C05483=1150.206,331.149,-77.116,-176.637,8.840,148.788
C05484=1150.202,331.397,-77.150,-176.634,8.844,148.788
C05485=1150.198,331.645,-77.183,-176.632,8.847,148.789
C05486=1150.193,331.893,-77.216,-176.629,8.851,148.789
C05487=1150.190,332.140,-77.248,-176.627,8.854,148.789
C05488=1150.186,332.388,-77.282,-176.624,8.858,148.789
C05489=1150.182,332.635,-77.315,-176.621,8.862,148.789
C05490=1150.178,332.883,-77.348,-176.619,8.865,148.790
C05491=1150.174,333.131,-77.381,-176.616,8.869,148.790
C05492=1150.169,333.379,-77.414,-176.614,8.872,148.790
C05493=1150.165,333.626,-77.447,-176.611,8.877,148.790
C05494=1150.161,333.874,-77.481,-176.609,8.880,148.791
C05495=1150.157,334.122,-77.514,-176.606,8.883,148.791
C05496=1150.153,334.370,-77.547,-176.603,8.887,148.791
C05497=1150.149,334.617,-77.580,-176.601,8.890,148.791
C05498=1150.145,334.865,-77.613,-176.599,8.895,148.792
C05499=1150.141,335.113,-77.647,-176.596,8.898,148.792
C05500=1150.137,335.361,-77.680,-176.593,8.902,148.792
C05501=1150.133,335.609,-77.713,-176.591,8.906,148.792
C05502=1150.129,335.856,-77.747,-176.589,8.909,148.792
C05503=1150.125,336.104,-77.780,-176.586,8.913,148.793
C05504=1150.121,336.351,-77.813,-176.583,8.916,148.793
C05505=1150.116,336.599,-77.846,-176.580,8.920,148.793
C05506=1150.112,336.847,-77.879,-176.578,8.924,148.793
C05507=1150.109,337.095,-77.913,-176.576,8.928,148.794
C05508=1150.105,337.342,-77.947,-176.573,8.931,148.794
C05509=1150.101,337.590,-77.980,-176.570,8.935,148.794
C05510=1150.097,337.838,-78.013,-176.568,8.939,148.794
C05511=1150.092,338.086,-78.047,-176.565,8.943,148.795
C05512=1150.088,338.333,-78.081,-176.563,8.946,148.795
C05513=1150.084,338.581,-78.114,-176.560,8.950,148.795
C05514=1150.080,338.829,-78.147,-176.558,8.953,148.795
C05515=1150.076,339.109,-78.185,-176.555,8.958,148.796
C05516=1150.071,339.389,-78.224,-176.552,8.962,148.796
C05517=1150.067,339.670,-78.261,-176.549,8.966,148.796
C05518=1150.062,339.950,-78.300,-176.547,8.970,148.797
C05519=1150.057,340.197,-78.333,-176.544,8.974,148.797
C05520=1150.054,340.445,-78.367,-176.541,8.977,148.797
C05521=1150.050,340.693,-78.400,-176.539,8.982,148.797
C05522=1150.046,340.940,-78.435,-176.536,8.985,148.798
C05523=1150.041,341.188,-78.468,-176.534,8.989,148.798
C05524=1150.038,341.436,-78.502,-176.531,8.992,148.798
C05525=1150.034,341.684,-78.535,-176.528,8.996,148.798
C05526=1150.029,341.931,-78.570,-176.526,9.000,148.799
C05527=1150.025,342.179,-78.603,-176.524,9.004,148.799
C05528=1150.022,342.427,-78.637,-176.521,9.007,148.799
C05529=1150.018,342.674,-78.670,-176.518,9.011,148.799
C05530=1150.013,342.922,-78.705,-176.516,9.015,148.800
C05531=1150.009,343.169,-78.738,-176.514,9.019,148.800
C05532=1150.006,343.417,-78.772,-176.511,9.022,148.800
C05533=1150.001,343.665,-78.806,-176.508,9.027,148.801
C05534=1149.997,343.912,-78.840,-176.506,9.030,148.801
C05535=1149.993,344.159,-78.873,-176.503,9.034,148.801
C05536=1149.989,344.408,-78.908,-176.501,9.037,148.801
C05537=1149.985,344.655,-78.941,-176.498,9.042,148.802
C05538=1149.981,344.903,-78.976,-176.496,9.045,148.802
C05539=1149.977,345.151,-79.009,-176.493,9.049,148.802
C05540=1149.973,345.398,-79.043,-176.491,9.052,148.803
C05541=1149.969,345.646,-79.078,-176.488,9.057,148.803
C05542=1149.965,345.894,-79.111,-176.486,9.060,148.803
C05543=1149.961,346.142,-79.146,-176.483,9.064,148.803
C05544=1149.957,346.389,-79.180,-176.481,9.068,148.804
C05545=1149.954,346.636,-79.214,-176.478,9.072,148.804
C05546=1149.949,346.884,-79.248,-176.476,9.075,148.804
C05547=1149.945,347.132,-79.281,-176.473,9.079,148.804
C05548=1149.941,347.380,-79.316,-176.471,9.083,148.805
C05549=1149.937,347.627,-79.350,-176.468,9.087,148.805
C05550=1149.933,347.875,-79.385,-176.466,9.090,148.805
C05551=1149.929,348.122,-79.419,-176.463,9.094,148.805
C05552=1149.925,348.370,-79.453,-176.461,9.098,148.806
C05553=1149.921,348.618,-79.487,-176.458,9.102,148.806
C05554=1149.917,348.865,-79.521,-176.455,9.106,148.806
C05555=1149.913,349.113,-79.556,-176.453,9.109,148.807
C05556=1149.909,349.361,-79.590,-176.450,9.113,148.807
C05557=1149.905,349.608,-79.624,-176.448,9.117,148.807
C05558=1149.901,349.856,-79.659,-176.445,9.121,148.808
C05559=1149.897,350.103,-79.693,-176.443,9.124,148.808
C05560=1149.893,350.351,-79.727,-176.440,9.128,148.808
C05561=1149.889,350.598,-79.761,-176.438,9.132,148.808
C05562=1149.886,350.846,-79.796,-176.436,9.136,148.809
C05563=1149.881,351.094,-79.831,-176.433,9.139,148.809
C05564=1149.878,351.341,-79.865,-176.430,9.144,148.809
C05565=1149.873,351.589,-79.899,-176.428,9.148,148.810
C05566=1149.869,351.836,-79.933,-176.426,9.151,148.810
C05567=1149.865,352.084,-79.968,-176.423,9.155,148.810
C05568=1149.861,352.332,-80.003,-176.421,9.159,148.811
C05569=1149.858,352.579,-80.037,-176.418,9.163,148.811
C05570=1149.853,352.826,-80.072,-176.416,9.166,148.811
C05571=1149.849,353.074,-80.107,-176.413,9.171,148.812
C05572=1149.845,353.321,-80.141,-176.410,9.175,148.812
C05573=1149.842,353.570,-80.175,-176.408,9.178,148.812
C05574=1149.837,353.817,-80.210,-176.405,9.182,148.813
C05575=1149.834,354.065,-80.244,-176.403,9.186,148.813
C05576=1149.830,354.312,-80.280,-176.400,9.190,148.813
C05577=1149.825,354.560,-80.314,-176.398,9.193,148.813
C05578=1149.822,354.808,-80.349,-176.395,9.197,148.814
C05579=1149.818,355.055,-80.383,-176.393,9.202,148.814
C05580=1149.814,355.302,-80.418,-176.391,9.205,148.814
C05581=1149.809,355.550,-80.453,-176.388,9.209,148.815
C05582=1149.806,355.798,-80.487,-176.386,9.213,148.815
C05583=1149.802,356.044,-80.522,-176.383,9.217,148.815
C05584=1149.798,356.293,-80.557,-176.380,9.221,148.816
C05585=1149.794,356.541,-80.592,-176.378,9.225,148.816
C05586=1149.790,356.787,-80.627,-176.375,9.229,148.816
C05587=1149.787,357.035,-80.661,-176.373,9.232,148.817
C05588=1149.782,357.282,-80.697,-176.370,9.236,148.817
C05589=1149.778,357.530,-80.731,-176.367,9.240,148.817
C05590=1149.774,357.778,-80.766,-176.365,9.244,148.818
C05591=1149.770,358.025,-80.801,-176.363,9.248,148.818
C05592=1149.767,358.273,-80.836,-176.361,9.252,148.818
C05593=1149.763,358.520,-80.871,-176.358,9.256,148.818
C05594=1149.759,358.768,-80.906,-176.355,9.260,148.819
C05595=1149.755,359.015,-80.941,-176.353,9.263,148.819
C05596=1149.750,359.263,-80.976,-176.350,9.267,148.819
C05597=1149.747,359.510,-81.011,-176.348,9.272,148.820
C05598=1149.743,359.758,-81.046,-176.345,9.275,148.820
C05599=1149.738,360.005,-81.081,-176.342,9.279,148.820
C05600=1149.735,360.253,-81.117,-176.340,9.284,148.821
C05601=1149.732,360.500,-81.151,-176.338,9.287,148.821
C05602=1149.727,360.747,-81.186,-176.335,9.291,148.821
C05603=1149.723,360.995,-81.221,-176.332,9.295,148.822
C05604=1149.720,361.243,-81.257,-176.330,9.299,148.822
C05605=1149.715,361.490,-81.292,-176.327,9.303,148.822
C05606=1149.711,361.738,-81.327,-176.324,9.307,148.823
C05607=1149.708,361.985,-81.362,-176.322,9.312,148.823
C05608=1149.704,362.233,-81.398,-176.320,9.315,148.823
C05609=1149.700,362.480,-81.433,-176.317,9.319,148.824
C05610=1149.696,362.728,-81.468,-176.314,9.323,148.824
C05611=1149.692,362.975,-81.503,-176.312,9.327,148.824
C05612=1149.688,363.222,-81.538,-176.309,9.331,148.825
C05613=1149.684,363.470,-81.574,-176.306,9.335,148.825
C05614=1149.680,363.718,-81.609,-176.304,9.339,148.825
C05615=1149.677,363.965,-81.644,-176.302,9.343,148.826
C05616=1149.673,364.213,-81.680,-176.299,9.347,148.826
C05617=1149.669,364.459,-81.715,-176.296,9.351,148.826
C05618=1149.665,364.707,-81.751,-176.293,9.355,148.827
C05619=1149.661,364.990,-81.791,-176.291,9.360,148.827
C05620=1149.656,365.274,-81.832,-176.287,9.365,148.828
C05621=1149.651,365.556,-81.873,-176.285,9.369,148.828
C05622=1149.646,365.840,-81.913,-176.281,9.374,148.828
C05623=1149.643,366.088,-81.948,-176.280,9.377,148.829
C05624=1149.639,366.335,-81.984,-176.277,9.382,148.829
C05625=1149.636,366.583,-82.019,-176.274,9.386,148.829
C05626=1149.631,366.830,-82.055,-176.271,9.390,148.830
C05627=1149.627,367.077,-82.091,-176.269,9.394,148.830
C05628=1149.623,367.325,-82.126,-176.266,9.398,148.830
C05629=1149.620,367.572,-82.162,-176.264,9.402,148.831
C05630=1149.616,367.820,-82.197,-176.261,9.407,148.831
C05631=1149.613,368.067,-82.234,-176.259,9.411,148.832
C05632=1149.608,368.314,-82.269,-176.257,9.414,148.832
C05633=1149.604,368.561,-82.305,-176.254,9.418,148.832
C05634=1149.600,368.809,-82.340,-176.251,9.423,148.833
C05635=1149.597,369.056,-82.376,-176.249,9.427,148.833
C05636=1149.592,369.304,-82.412,-176.246,9.430,148.833
C05637=1149.588,369.552,-82.448,-176.244,9.435,148.834
C05638=1149.585,369.799,-82.483,-176.241,9.439,148.834
C05639=1149.581,370.046,-82.520,-176.239,9.443,148.835
C05640=1149.576,370.293,-82.555,-176.236,9.448,148.835
C05641=1149.573,370.541,-82.591,-176.234,9.451,148.836
C05642=1149.569,370.788,-82.626,-176.232,9.456,148.836
C05643=1149.565,371.036,-82.663,-176.229,9.460,148.837
C05644=1149.561,371.283,-82.699,-176.226,9.464,148.837
C05645=1149.558,371.530,-82.734,-176.224,9.468,148.837
C05646=1149.553,371.778,-82.770,-176.222,9.472,148.838
C05647=1149.550,372.025,-82.807,-176.219,9.476,148.838
C05648=1149.546,372.273,-82.843,-176.217,9.480,148.839
C05649=1149.542,372.520,-82.878,-176.215,9.484,148.839
C05650=1149.539,372.767,-82.915,-176.212,9.489,148.840
C05651=1149.534,373.015,-82.951,-176.211,9.492,148.840
C05652=1149.530,373.263,-82.986,-176.208,9.497,148.840
C05653=1149.527,373.510,-83.023,-176.206,9.501,148.841
C05654=1149.523,373.757,-83.059,-176.204,9.505,148.841
C05655=1149.519,374.004,-83.095,-176.201,9.509,148.842
C05656=1149.515,374.252,-83.131,-176.199,9.514,148.842
C05657=1149.511,374.498,-83.167,-176.197,9.517,148.843
C05658=1149.507,374.746,-83.203,-176.195,9.522,148.843
C05659=1149.503,374.994,-83.239,-176.193,9.525,148.844
C05660=1149.499,375.241,-83.276,-176.191,9.530,148.844
C05661=1149.495,375.488,-83.311,-176.189,9.534,148.845
C05662=1149.492,375.736,-83.348,-176.186,9.538,148.845
C05663=1149.488,375.983,-83.385,-176.185,9.542,148.846
C05664=1149.484,376.231,-83.421,-176.182,9.546,148.846
C05665=1149.481,376.478,-83.457,-176.181,9.550,148.847
C05666=1149.476,376.726,-83.493,-176.178,9.555,148.848
C05667=1149.473,376.972,-83.529,-176.177,9.559,148.848
C05668=1149.468,377.220,-83.566,-176.175,9.562,148.849
C05669=1149.465,377.467,-83.602,-176.173,9.567,148.849
C05670=1149.461,377.714,-83.639,-176.172,9.571,148.850
C05671=1149.457,377.962,-83.674,-176.170,9.574,148.850
C05672=1149.453,378.209,-83.711,-176.168,9.579,148.851
C05673=1149.449,378.456,-83.748,-176.166,9.583,148.852
C05674=1149.445,378.704,-83.784,-176.165,9.587,148.852
C05675=1149.441,378.951,-83.820,-176.163,9.591,148.853
C05676=1149.438,379.198,-83.857,-176.162,9.595,148.853
C05677=1149.434,379.446,-83.893,-176.160,9.598,148.854
C05678=1149.429,379.693,-83.930,-176.159,9.602,148.855
C05679=1149.426,379.940,-83.966,-176.157,9.607,148.855
C05680=1149.422,380.187,-84.003,-176.155,9.611,148.856
C05681=1149.419,380.435,-84.039,-176.154,9.614,148.856
C05682=1149.415,380.682,-84.076,-176.153,9.618,148.857
C05683=1149.411,380.929,-84.112,-176.152,9.622,148.858
C05684=1149.407,381.176,-84.149,-176.150,9.626,148.859
C05685=1149.403,381.423,-84.186,-176.149,9.630,148.859
C05686=1149.399,381.671,-84.222,-176.148,9.634,148.860
C05687=1149.396,381.918,-84.258,-176.147,9.637,148.861
C05688=1149.391,382.165,-84.295,-176.146,9.641,148.861
C05689=1149.387,382.413,-84.332,-176.145,9.644,148.862
C05690=1149.385,382.660,-84.368,-176.144,9.649,148.863
C05691=1149.381,382.907,-84.405,-176.143,9.652,148.863
C05692=1149.376,383.154,-84.442,-176.142,9.656,148.864
C05693=1149.372,383.402,-84.478,-176.141,9.659,148.865
C05694=1149.369,383.649,-84.514,-176.140,9.663,148.866
C05695=1149.365,383.896,-84.551,-176.140,9.667,148.866
C05696=1149.360,384.144,-84.588,-176.139,9.670,148.867
C05697=1149.358,384.391,-84.625,-176.138,9.673,148.868
C05698=1149.354,384.638,-84.662,-176.138,9.677,148.868
C05699=1149.350,384.886,-84.699,-176.137,9.680,148.869
C05700=1149.345,385.133,-84.735,-176.137,9.684,148.870
C05701=1149.342,385.380,-84.772,-176.137,9.687,148.871
C05702=1149.338,385.627,-84.808,-176.136,9.690,148.872
C05703=1149.335,385.875,-84.846,-176.136,9.694,148.872
C05704=1149.330,386.122,-84.883,-176.136,9.696,148.873
C05705=1149.327,386.369,-84.919,-176.136,9.700,148.874
C05706=1149.323,386.616,-84.956,-176.136,9.703,148.875
C05707=1149.319,386.863,-84.993,-176.136,9.706,148.876
C05708=1149.315,387.111,-85.030,-176.136,9.710,148.877
C05709=1149.311,387.358,-85.067,-176.136,9.712,148.877
C05710=1149.308,387.605,-85.103,-176.136,9.715,148.878
C05711=1149.304,387.852,-85.140,-176.136,9.719,148.879
C05712=1149.300,388.099,-85.177,-176.136,9.721,148.880
C05713=1149.296,388.347,-85.214,-176.136,9.724,148.880
C05714=1149.293,388.594,-85.250,-176.137,9.727,148.881
C05715=1149.289,388.841,-85.287,-176.136,9.730,148.882
C05716=1149.285,389.089,-85.324,-176.137,9.733,148.883
C05717=1149.281,389.336,-85.361,-176.138,9.736,148.884
C05718=1149.277,389.584,-85.398,-176.138,9.739,148.885
C05719=1149.274,389.831,-85.434,-176.138,9.741,148.886
C05720=1149.270,390.078,-85.471,-176.139,9.744,148.886
C05721=1149.266,390.325,-85.508,-176.139,9.747,148.887
C05722=1149.261,390.572,-85.545,-176.140,9.749,148.888
C05723=1149.257,390.858,-85.588,-176.141,9.752,148.889
C05724=1149.253,391.145,-85.630,-176.141,9.755,148.890
C05725=1149.249,391.432,-85.673,-176.142,9.758,148.891
C05726=1149.244,391.718,-85.716,-176.143,9.761,148.892
C05727=1149.241,391.966,-85.753,-176.143,9.764,148.893
C05728=1149.237,392.213,-85.790,-176.144,9.767,148.894
C05729=1149.233,392.460,-85.827,-176.145,9.769,148.895
C05730=1149.229,392.707,-85.863,-176.145,9.771,148.895
C05731=1149.225,392.955,-85.900,-176.146,9.773,148.896
C05732=1149.222,393.202,-85.937,-176.147,9.776,148.897
C05733=1149.218,393.449,-85.974,-176.148,9.778,148.898
C05734=1149.214,393.696,-86.011,-176.148,9.781,148.899
C05735=1149.210,393.943,-86.048,-176.149,9.783,148.900
C05736=1149.206,394.191,-86.085,-176.151,9.785,148.900
C05737=1149.202,394.438,-86.122,-176.151,9.788,148.901
C05738=1149.199,394.685,-86.159,-176.152,9.790,148.902
C05739=1149.195,394.932,-86.195,-176.153,9.792,148.903
C05740=1149.191,395.180,-86.232,-176.153,9.795,148.904
C05741=1149.187,395.427,-86.269,-176.155,9.797,148.905
C05742=1149.183,395.675,-86.306,-176.156,9.799,148.905
C05743=1149.179,395.922,-86.343,-176.157,9.801,148.906
C05744=1149.175,396.168,-86.381,-176.157,9.804,148.907
C05745=1149.172,396.415,-86.417,-176.158,9.806,148.908
C05746=1149.168,396.663,-86.454,-176.160,9.808,148.909
C05747=1149.164,396.910,-86.491,-176.161,9.810,148.910
C05748=1149.160,397.158,-86.528,-176.162,9.812,148.910
C05749=1149.156,397.405,-86.565,-176.163,9.814,148.911
C05750=1149.153,397.653,-86.602,-176.164,9.816,148.912
C05751=1149.149,397.899,-86.638,-176.165,9.818,148.913
C05752=1149.145,398.147,-86.675,-176.166,9.820,148.914
C05753=1149.141,398.393,-86.713,-176.167,9.822,148.914
C05754=1149.137,398.640,-86.750,-176.167,9.825,148.915
C05755=1149.134,398.888,-86.787,-176.168,9.827,148.916
C05756=1149.130,399.135,-86.824,-176.170,9.829,148.917
C05757=1149.126,399.383,-86.861,-176.171,9.831,148.918
C05758=1149.122,399.630,-86.897,-176.172,9.833,148.919
C05759=1149.119,399.877,-86.934,-176.172,9.835,148.919
C05760=1149.115,400.125,-86.971,-176.174,9.836,148.920
C05761=1149.111,400.372,-87.008,-176.175,9.838,148.921
C05762=1149.107,400.618,-87.045,-176.176,9.840,148.922
C05763=1149.103,400.866,-87.082,-176.177,9.843,148.923
C05764=1149.099,401.113,-87.119,-176.179,9.845,148.923
C05765=1149.096,401.360,-87.156,-176.179,9.846,148.924
C05766=1149.092,401.608,-87.193,-176.180,9.848,148.925
C05767=1149.088,401.855,-87.229,-176.181,9.850,148.926
C05768=1149.084,402.102,-87.266,-176.183,9.853,148.927
C05769=1149.080,402.350,-87.303,-176.183,9.854,148.927
C05770=1149.076,402.596,-87.341,-176.184,9.856,148.928
C05771=1149.072,402.844,-87.378,-176.185,9.858,148.929
C05772=1149.069,403.090,-87.414,-176.187,9.860,148.930
C05773=1149.065,403.338,-87.451,-176.187,9.862,148.930
C05774=1149.061,403.586,-87.488,-176.189,9.863,148.931
C05775=1149.057,403.833,-87.525,-176.190,9.866,148.932
C05776=1149.053,404.080,-87.562,-176.191,9.867,148.933
C05777=1149.049,404.327,-87.599,-176.192,9.869,148.933
C05778=1149.045,404.575,-87.636,-176.193,9.871,148.934
C05779=1149.042,404.821,-87.673,-176.194,9.873,148.935
C05780=1149.038,405.068,-87.710,-176.195,9.875,148.936
C05781=1149.034,405.316,-87.747,-176.196,9.877,148.937
C05782=1149.031,405.564,-87.784,-176.196,9.879,148.937
C05783=1149.027,405.811,-87.821,-176.198,9.881,148.938
C05784=1149.023,406.058,-87.858,-176.199,9.882,148.939
C05785=1149.018,406.305,-87.895,-176.200,9.884,148.940
C05786=1149.015,406.552,-87.931,-176.201,9.886,148.940
C05787=1149.012,406.799,-87.969,-176.202,9.888,148.941
C05788=1149.008,407.046,-88.006,-176.203,9.890,148.942
C05789=1149.004,407.294,-88.042,-176.203,9.892,148.942
C05790=1149.000,407.541,-88.079,-176.205,9.894,148.943
C05791=1148.996,407.789,-88.117,-176.205,9.896,148.944
C05792=1148.992,408.036,-88.153,-176.206,9.898,148.945
C05793=1148.989,408.283,-88.190,-176.207,9.899,148.945
C05794=1148.985,408.530,-88.227,-176.208,9.901,148.946
C05795=1148.981,408.777,-88.264,-176.209,9.903,148.947
C05796=1148.977,409.024,-88.301,-176.209,9.905,148.948
C05797=1148.973,409.272,-88.338,-176.211,9.907,148.948
C05798=1148.969,409.519,-88.375,-176.211,9.909,148.949
C05799=1148.965,409.766,-88.412,-176.212,9.911,148.950
C05800=1148.962,410.014,-88.449,-176.213,9.913,148.951
C05801=1148.958,410.261,-88.485,-176.214,9.914,148.951
C05802=1148.954,410.508,-88.522,-176.215,9.916,148.952
C05803=1148.950,410.755,-88.560,-176.215,9.918,148.953
C05804=1148.947,411.002,-88.597,-176.216,9.920,148.953
C05805=1148.943,411.250,-88.634,-176.217,9.922,148.954
C05806=1148.939,411.497,-88.671,-176.218,9.924,148.955
C05807=1148.934,411.744,-88.708,-176.219,9.925,148.955
C05808=1148.931,411.991,-88.744,-176.220,9.928,148.956
C05809=1148.928,412.239,-88.781,-176.220,9.929,148.957
C05810=1148.924,412.485,-88.819,-176.221,9.931,148.957
C05811=1148.920,412.733,-88.856,-176.222,9.933,148.958
C05812=1148.916,412.980,-88.892,-176.223,9.935,148.959
C05813=1148.912,413.228,-88.930,-176.223,9.937,148.960
C05814=1148.908,413.475,-88.966,-176.224,9.939,148.960
C05815=1148.904,413.722,-89.003,-176.225,9.941,148.961
C05816=1148.901,413.969,-89.040,-176.225,9.943,148.962
C05817=1148.897,414.215,-89.077,-176.226,9.945,148.962
C05818=1148.893,414.463,-89.114,-176.227,9.946,148.963
C05819=1148.889,414.711,-89.151,-176.228,9.949,148.964
C05820=1148.886,414.958,-89.188,-176.228,9.950,148.965
C05821=1148.883,415.204,-89.225,-176.228,9.953,148.965
C05822=1148.881,415.453,-89.262,-176.229,9.955,148.966
C05823=1148.881,415.679,-89.296,-176.230,9.956,148.966
C05824=1148.880,415.906,-89.329,-176.231,9.958,148.967
C05825=1148.880,416.132,-89.362,-176.231,9.960,148.968
C05826=1148.881,416.359,-89.396,-176.231,9.961,148.968
C05827=1148.882,416.585,-89.429,-176.232,9.963,148.969
C05828=1148.885,416.812,-89.463,-176.233,9.965,148.969
C05829=1148.887,417.038,-89.495,-176.233,9.966,148.970
C05830=1148.891,417.263,-89.528,-176.234,9.968,148.971
C05831=1148.470,417.266,-89.578,-176.236,9.979,148.974
C05832=1148.467,417.038,-89.545,-176.236,9.977,148.973
C05833=1148.464,416.810,-89.511,-176.235,9.975,148.973
C05834=1148.462,416.582,-89.478,-176.235,9.974,148.972
C05835=1148.460,416.354,-89.444,-176.234,9.972,148.972
C05836=1148.460,416.126,-89.410,-176.233,9.970,148.971
C05837=1148.460,415.897,-89.376,-176.233,9.969,148.971
C05838=1148.460,415.669,-89.342,-176.232,9.967,148.970
C05839=1148.461,415.441,-89.309,-176.232,9.965,148.969
C05840=1148.463,415.194,-89.272,-176.231,9.964,148.969
C05841=1148.465,414.946,-89.236,-176.230,9.962,148.968
C05842=1148.469,414.699,-89.198,-176.229,9.960,148.967
C05843=1148.473,414.452,-89.161,-176.229,9.958,148.967
C05844=1148.476,414.204,-89.124,-176.229,9.955,148.966
C05845=1148.480,413.957,-89.087,-176.228,9.954,148.965
C05846=1148.484,413.710,-89.051,-176.227,9.952,148.964
C05847=1148.488,413.463,-89.014,-176.226,9.950,148.964
C05848=1148.492,413.216,-88.976,-176.225,9.948,148.963
C05849=1148.495,412.968,-88.939,-176.224,9.946,148.962
C05850=1148.499,412.721,-88.902,-176.224,9.944,148.962
C05851=1148.503,412.474,-88.865,-176.223,9.943,148.961
C05852=1148.507,412.227,-88.828,-176.223,9.940,148.960
C05853=1148.510,411.979,-88.792,-176.222,9.938,148.960
C05854=1148.514,411.732,-88.755,-176.221,9.936,148.959
C05855=1148.518,411.485,-88.717,-176.221,9.934,148.958
C05856=1148.522,411.238,-88.680,-176.219,9.932,148.957
C05857=1148.526,410.990,-88.643,-176.219,9.931,148.957
C05858=1148.530,410.743,-88.606,-176.218,9.929,148.956
C05859=1148.534,410.496,-88.569,-176.217,9.927,148.955
C05860=1148.538,410.249,-88.533,-176.216,9.925,148.955
C05861=1148.541,410.003,-88.496,-176.215,9.923,148.954
C05862=1148.544,409.755,-88.458,-176.215,9.921,148.953
C05863=1148.548,409.507,-88.422,-176.213,9.919,148.952
C05864=1148.553,409.260,-88.385,-176.213,9.917,148.952
C05865=1148.557,409.013,-88.348,-176.212,9.916,148.951
C05866=1148.560,408.765,-88.311,-176.211,9.914,148.950
C05867=1148.564,408.518,-88.274,-176.210,9.912,148.950
C05868=1148.568,408.271,-88.236,-176.209,9.910,148.949
C05869=1148.571,408.025,-88.200,-176.209,9.908,148.948
C05870=1148.575,407.777,-88.163,-176.207,9.906,148.947
C05871=1148.579,407.530,-88.126,-176.207,9.904,148.947
C05872=1148.583,407.282,-88.089,-176.206,9.902,148.946
C05873=1148.587,407.035,-88.052,-176.205,9.900,148.945
C05874=1148.591,406.788,-88.015,-176.203,9.899,148.944
C05875=1148.595,406.540,-87.978,-176.202,9.897,148.944
C05876=1148.598,406.294,-87.941,-176.202,9.895,148.943
C05877=1148.602,406.047,-87.904,-176.200,9.893,148.942
C05878=1148.606,405.799,-87.867,-176.200,9.891,148.941
C05879=1148.610,405.552,-87.830,-176.199,9.889,148.941
C05880=1148.614,405.304,-87.793,-176.198,9.887,148.940
C05881=1148.618,405.057,-87.756,-176.197,9.886,148.939
C05882=1148.622,404.810,-87.720,-176.196,9.884,148.938
C05883=1148.626,404.563,-87.682,-176.195,9.881,148.937
C05884=1148.628,404.316,-87.645,-176.193,9.881,148.937
C05885=1148.632,404.069,-87.608,-176.192,9.878,148.936
C05886=1148.637,403.821,-87.572,-176.191,9.876,148.935
C05887=1148.641,403.574,-87.535,-176.191,9.875,148.935
C05888=1148.644,403.326,-87.498,-176.189,9.873,148.934
C05889=1148.648,403.079,-87.461,-176.188,9.871,148.933
C05890=1148.652,402.833,-87.423,-176.188,9.869,148.932
C05891=1148.655,402.586,-87.387,-176.187,9.867,148.931
C05892=1148.659,402.338,-87.350,-176.185,9.865,148.931
C05893=1148.663,402.091,-87.313,-176.184,9.863,148.930
C05894=1148.667,401.843,-87.276,-176.183,9.861,148.929
C05895=1148.671,401.596,-87.239,-176.182,9.860,148.928
C05896=1148.675,401.349,-87.202,-176.181,9.858,148.927
C05897=1148.679,401.101,-87.165,-176.180,9.855,148.927
C05898=1148.682,400.855,-87.128,-176.179,9.853,148.926
C05899=1148.686,400.608,-87.091,-176.178,9.851,148.925
C05900=1148.690,400.361,-87.054,-176.177,9.850,148.924
C05901=1148.693,400.113,-87.017,-176.176,9.848,148.923
C05902=1148.698,399.865,-86.980,-176.175,9.845,148.923
C05903=1148.702,399.618,-86.943,-176.174,9.843,148.922
C05904=1148.706,399.371,-86.906,-176.172,9.841,148.921
C05905=1148.709,399.124,-86.870,-176.171,9.839,148.920
C05906=1148.712,398.877,-86.832,-176.170,9.837,148.919
C05907=1148.716,398.630,-86.795,-176.169,9.835,148.918
C05908=1148.720,398.383,-86.759,-176.168,9.833,148.918
C05909=1148.725,398.135,-86.722,-176.167,9.831,148.917
C05910=1148.728,397.887,-86.684,-176.166,9.829,148.916
C05911=1148.732,397.640,-86.648,-176.165,9.827,148.915
C05912=1148.736,397.393,-86.611,-176.164,9.825,148.914
C05913=1148.740,397.146,-86.574,-176.163,9.823,148.914
C05914=1148.743,396.900,-86.537,-176.162,9.821,148.913
C05915=1148.747,396.652,-86.500,-176.161,9.819,148.912
C05916=1148.751,396.405,-86.463,-176.160,9.816,148.911
C05917=1148.755,396.157,-86.426,-176.159,9.814,148.910
C05918=1148.759,395.910,-86.389,-176.158,9.812,148.909
C05919=1148.763,395.662,-86.352,-176.157,9.810,148.909
C05920=1148.766,395.415,-86.316,-176.156,9.808,148.908
C05921=1148.770,395.168,-86.279,-176.156,9.805,148.907
C05922=1148.774,394.922,-86.241,-176.155,9.803,148.906
C05923=1148.778,394.674,-86.204,-176.153,9.801,148.905
C05924=1148.781,394.427,-86.167,-176.152,9.799,148.904
C05925=1148.786,394.179,-86.130,-176.152,9.796,148.904
C05926=1148.789,393.932,-86.094,-176.151,9.794,148.903
C05927=1148.793,393.685,-86.057,-176.150,9.792,148.902
C05928=1148.797,393.437,-86.020,-176.149,9.789,148.901
C05929=1148.801,393.190,-85.983,-176.148,9.787,148.900
C05930=1148.805,392.943,-85.946,-176.147,9.784,148.899
C05931=1148.809,392.696,-85.909,-176.147,9.783,148.899
C05932=1148.813,392.449,-85.872,-176.146,9.780,148.898
C05933=1148.815,392.202,-85.835,-176.145,9.778,148.897
C05934=1148.819,391.954,-85.798,-176.145,9.775,148.896
C05935=1148.824,391.707,-85.761,-176.144,9.772,148.895
C05936=1148.828,391.420,-85.719,-176.144,9.769,148.894
C05937=1148.832,391.134,-85.676,-176.143,9.766,148.893
C05938=1148.837,390.847,-85.633,-176.142,9.763,148.892
C05939=1148.841,390.561,-85.590,-176.141,9.760,148.891
C05940=1148.845,390.314,-85.553,-176.140,9.758,148.891
C05941=1148.848,390.066,-85.516,-176.140,9.755,148.890
C05942=1148.852,389.819,-85.480,-176.139,9.752,148.889
C05943=1148.856,389.572,-85.443,-176.139,9.750,148.888
C05944=1148.860,389.325,-85.406,-176.139,9.747,148.887
C05945=1148.864,389.077,-85.369,-176.138,9.744,148.886
C05946=1148.867,388.830,-85.332,-176.138,9.741,148.886
C05947=1148.871,388.583,-85.296,-176.138,9.739,148.885
C05948=1148.875,388.336,-85.259,-176.138,9.735,148.884
C05949=1148.880,388.088,-85.222,-176.138,9.732,148.883
C05950=1148.883,387.841,-85.185,-176.137,9.729,148.882
C05951=1148.886,387.594,-85.148,-176.137,9.727,148.881
C05952=1148.891,387.346,-85.111,-176.137,9.723,148.880
C05953=1148.895,387.099,-85.075,-176.137,9.721,148.880
C05954=1148.899,386.852,-85.038,-176.137,9.717,148.879
C05955=1148.902,386.604,-85.001,-176.137,9.714,148.878
C05956=1148.906,386.357,-84.964,-176.137,9.711,148.877
C05957=1148.910,386.110,-84.927,-176.137,9.708,148.877
C05958=1148.914,385.863,-84.891,-176.137,9.705,148.876
C05959=1148.918,385.616,-84.854,-176.138,9.701,148.875
C05960=1148.921,385.369,-84.817,-176.138,9.698,148.874
C05961=1148.925,385.121,-84.780,-176.139,9.695,148.873
C05962=1148.929,384.874,-84.743,-176.139,9.691,148.873
C05963=1148.933,384.627,-84.706,-176.140,9.688,148.872
C05964=1148.936,384.380,-84.670,-176.140,9.684,148.871
C05965=1148.940,384.133,-84.633,-176.141,9.681,148.870
C05966=1148.944,383.885,-84.597,-176.141,9.678,148.870
C05967=1148.948,383.637,-84.559,-176.142,9.674,148.869
C05968=1148.951,383.391,-84.523,-176.143,9.670,148.868
C05969=1148.955,383.143,-84.486,-176.144,9.667,148.867
C05970=1148.959,382.896,-84.449,-176.144,9.664,148.867
C05971=1148.963,382.649,-84.413,-176.145,9.659,148.866
C05972=1148.967,382.401,-84.377,-176.146,9.656,148.865
C05973=1148.971,382.154,-84.340,-176.147,9.652,148.865
C05974=1148.975,381.906,-84.303,-176.149,9.648,148.864
C05975=1148.978,381.660,-84.267,-176.149,9.645,148.863
C05976=1148.982,381.412,-84.230,-176.150,9.641,148.863
C05977=1148.986,381.165,-84.193,-176.152,9.637,148.862
C05978=1148.990,380.918,-84.157,-176.153,9.633,148.861
C05979=1148.994,380.670,-84.120,-176.155,9.629,148.860
C05980=1148.998,380.423,-84.084,-176.155,9.626,148.860
C05981=1149.002,380.176,-84.047,-176.157,9.622,148.859
C05982=1149.005,379.928,-84.010,-176.158,9.618,148.858
C05983=1149.009,379.681,-83.975,-176.159,9.614,148.858
C05984=1149.013,379.434,-83.938,-176.161,9.610,148.857
C05985=1149.017,379.187,-83.901,-176.163,9.605,148.857
C05986=1149.020,378.940,-83.865,-176.164,9.602,148.856
C05987=1149.025,378.692,-83.828,-176.166,9.598,148.856
C05988=1149.029,378.445,-83.792,-176.168,9.594,148.855
C05989=1149.032,378.198,-83.755,-176.169,9.590,148.854
C05990=1149.037,377.950,-83.719,-176.171,9.586,148.854
C05991=1149.040,377.703,-83.683,-176.173,9.582,148.853
C05992=1149.044,377.456,-83.646,-176.175,9.578,148.853
C05993=1149.048,377.208,-83.610,-176.177,9.573,148.852
C05994=1149.052,376.961,-83.574,-176.179,9.570,148.852
C05995=1149.056,376.713,-83.537,-176.180,9.566,148.851
C05996=1149.059,376.467,-83.501,-176.183,9.561,148.850
C05997=1149.064,376.219,-83.464,-176.184,9.558,148.850
C05998=1149.067,375.972,-83.429,-176.187,9.553,148.849
C05999=1149.071,375.724,-83.392,-176.188,9.549,148.849
C06000=1149.074,375.476,-83.356,-176.191,9.545,148.848
C06001=1149.078,375.229,-83.319,-176.193,9.541,148.848
C06002=1149.082,374.982,-83.284,-176.195,9.537,148.847
C06003=1149.086,374.735,-83.247,-176.197,9.533,148.847
C06004=1149.090,374.487,-83.211,-176.199,9.529,148.846
C06005=1149.093,374.240,-83.175,-176.202,9.524,148.846
C06006=1149.098,373.992,-83.139,-176.203,9.520,148.845
C06007=1149.101,373.746,-83.103,-176.205,9.516,148.845
C06008=1149.106,373.498,-83.067,-176.207,9.512,148.844
C06009=1149.109,373.252,-83.031,-176.210,9.508,148.844
C06010=1149.114,373.004,-82.994,-176.212,9.504,148.843
C06011=1149.117,372.756,-82.959,-176.215,9.499,148.843
C06012=1149.121,372.509,-82.923,-176.217,9.496,148.842
C06013=1149.125,372.262,-82.886,-176.219,9.491,148.842
C06014=1149.129,372.014,-82.851,-176.222,9.487,148.842
C06015=1149.132,371.767,-82.815,-176.224,9.483,148.841
C06016=1149.137,371.519,-82.778,-176.227,9.479,148.841
C06017=1149.140,371.272,-82.743,-176.229,9.475,148.840
C06018=1149.144,371.025,-82.706,-176.232,9.470,148.840
C06019=1149.148,370.777,-82.671,-176.233,9.467,148.839
C06020=1149.152,370.530,-82.635,-176.236,9.462,148.839
C06021=1149.155,370.282,-82.599,-176.239,9.458,148.839
C06022=1149.159,370.035,-82.563,-176.241,9.454,148.838
C06023=1149.164,369.788,-82.527,-176.243,9.450,148.838
C06024=1149.167,369.541,-82.492,-176.246,9.446,148.837
C06025=1149.172,369.293,-82.456,-176.249,9.442,148.837
C06026=1149.175,369.045,-82.420,-176.251,9.437,148.837
C06027=1149.179,368.798,-82.385,-176.254,9.433,148.836
C06028=1149.183,368.550,-82.349,-176.256,9.430,148.836
C06029=1149.187,368.303,-82.312,-176.258,9.425,148.835
C06030=1149.191,368.056,-82.277,-176.261,9.421,148.835
C06031=1149.195,367.809,-82.241,-176.264,9.417,148.835
C06032=1149.198,367.561,-82.206,-176.266,9.413,148.834
C06033=1149.203,367.314,-82.170,-176.269,9.409,148.834
C06034=1149.207,367.066,-82.134,-176.271,9.405,148.834
C06035=1149.210,366.819,-82.099,-176.274,9.401,148.833
C06036=1149.214,366.571,-82.063,-176.276,9.396,148.833
C06037=1149.218,366.324,-82.028,-176.279,9.392,148.833
C06038=1149.222,366.077,-81.992,-176.281,9.389,148.832
C06039=1149.226,365.829,-81.956,-176.284,9.385,148.832
C06040=1149.230,365.546,-81.916,-176.287,9.379,148.831
C06041=1149.234,365.263,-81.875,-176.290,9.375,148.831
C06042=1149.239,364.980,-81.835,-176.293,9.371,148.831
C06043=1149.244,364.696,-81.794,-176.296,9.366,148.830
C06044=1149.248,364.448,-81.759,-176.299,9.362,148.830
C06045=1149.251,364.201,-81.724,-176.301,9.358,148.830
C06046=1149.255,363.953,-81.688,-176.303,9.354,148.829
C06047=1149.259,363.707,-81.653,-176.306,9.350,148.829
C06048=1149.263,363.459,-81.617,-176.309,9.345,148.828
C06049=1149.267,363.212,-81.582,-176.312,9.341,148.828
C06050=1149.271,362.963,-81.547,-176.314,9.338,148.828
C06051=1149.275,362.717,-81.512,-176.317,9.334,148.827
C06052=1149.278,362.469,-81.476,-176.320,9.330,148.827
C06053=1149.282,362.222,-81.441,-176.321,9.326,148.827
C06054=1149.286,361.974,-81.406,-176.324,9.322,148.827
C06055=1149.290,361.727,-81.371,-176.327,9.318,148.826
C06056=1149.294,361.479,-81.335,-176.330,9.313,148.826
C06057=1149.298,361.231,-81.300,-176.332,9.310,148.826
C06058=1149.302,360.984,-81.265,-176.335,9.306,148.825
C06059=1149.306,360.737,-81.230,-176.337,9.302,148.825
C06060=1149.310,360.489,-81.195,-176.340,9.298,148.825
C06061=1149.314,360.242,-81.160,-176.342,9.294,148.824
C06062=1149.318,359.994,-81.124,-176.345,9.290,148.824
C06063=1149.322,359.746,-81.089,-176.347,9.286,148.824
C06064=1149.326,359.499,-81.054,-176.350,9.282,148.823
C06065=1149.330,359.251,-81.019,-176.352,9.278,148.823
C06066=1149.334,359.004,-80.984,-176.355,9.275,148.823
C06067=1149.338,358.757,-80.950,-176.358,9.271,148.822
C06068=1149.341,358.509,-80.914,-176.360,9.266,148.822
C06069=1149.345,358.261,-80.879,-176.363,9.263,148.822
C06070=1149.349,358.014,-80.844,-176.365,9.258,148.821
C06071=1149.353,357.766,-80.809,-176.368,9.254,148.821
C06072=1149.357,357.519,-80.774,-176.370,9.251,148.821
C06073=1149.362,357.271,-80.739,-176.373,9.247,148.820
C06074=1149.365,357.024,-80.704,-176.375,9.243,148.820
C06075=1149.369,356.777,-80.670,-176.378,9.239,148.820
C06076=1149.373,356.529,-80.635,-176.380,9.235,148.819
C06077=1149.377,356.281,-80.600,-176.383,9.232,148.819
C06078=1149.381,356.034,-80.565,-176.385,9.227,148.819
C06079=1149.385,355.786,-80.531,-176.388,9.223,148.818
C06080=1149.389,355.539,-80.496,-176.390,9.220,148.818
C06081=1149.393,355.291,-80.461,-176.393,9.216,148.818
C06082=1149.397,355.043,-80.426,-176.395,9.212,148.817
C06083=1149.400,354.796,-80.391,-176.398,9.208,148.817
C06084=1149.405,354.549,-80.357,-176.400,9.205,148.817
C06085=1149.409,354.301,-80.322,-176.403,9.200,148.817
C06086=1149.412,354.053,-80.288,-176.405,9.196,148.816
C06087=1149.416,353.806,-80.253,-176.408,9.193,148.816
C06088=1149.420,353.558,-80.218,-176.411,9.189,148.816
C06089=1149.424,353.311,-80.184,-176.413,9.185,148.815
C06090=1149.428,353.063,-80.149,-176.416,9.181,148.815
C06091=1149.433,352.815,-80.115,-176.418,9.177,148.815
C06092=1149.436,352.568,-80.081,-176.420,9.173,148.814
C06093=1149.440,352.321,-80.045,-176.423,9.169,148.814
C06094=1149.444,352.073,-80.011,-176.425,9.166,148.814
C06095=1149.448,351.826,-79.977,-176.428,9.162,148.813
C06096=1149.452,351.577,-79.942,-176.430,9.158,148.813
C06097=1149.456,351.330,-79.907,-176.433,9.154,148.813
C06098=1149.460,351.082,-79.873,-176.436,9.150,148.812
C06099=1149.464,350.835,-79.839,-176.438,9.147,148.812
C06100=1149.468,350.588,-79.805,-176.441,9.142,148.812
C06101=1149.472,350.340,-79.770,-176.443,9.139,148.812
C06102=1149.477,350.092,-79.735,-176.446,9.135,148.811
C06103=1149.480,349.844,-79.701,-176.448,9.132,148.811
C06104=1149.484,349.597,-79.667,-176.451,9.127,148.811
C06105=1149.488,349.349,-79.633,-176.453,9.124,148.810
C06106=1149.492,349.102,-79.598,-176.456,9.120,148.810
C06107=1149.496,348.855,-79.564,-176.458,9.116,148.810
C06108=1149.500,348.606,-79.529,-176.461,9.112,148.810
C06109=1149.504,348.359,-79.495,-176.464,9.108,148.809
C06110=1149.508,348.111,-79.461,-176.465,9.104,148.809
C06111=1149.512,347.863,-79.427,-176.468,9.100,148.809
C06112=1149.517,347.616,-79.393,-176.471,9.097,148.808
C06113=1149.520,347.368,-79.359,-176.474,9.093,148.808
C06114=1149.524,347.121,-79.324,-176.475,9.089,148.808
C06115=1149.528,346.873,-79.290,-176.478,9.085,148.807
C06116=1149.532,346.626,-79.256,-176.481,9.082,148.807
C06117=1149.536,346.378,-79.222,-176.483,9.078,148.807
C06118=1149.540,346.130,-79.188,-176.485,9.074,148.807
C06119=1149.544,345.883,-79.154,-176.488,9.070,148.806
C06120=1149.548,345.636,-79.120,-176.491,9.067,148.806
C06121=1149.552,345.387,-79.086,-176.493,9.063,148.806
C06122=1149.556,345.140,-79.052,-176.496,9.059,148.806
C06123=1149.561,344.892,-79.017,-176.498,9.055,148.805
C06124=1149.564,344.644,-78.984,-176.501,9.051,148.805
C06125=1149.568,344.397,-78.950,-176.504,9.048,148.805
C06126=1149.573,344.149,-78.916,-176.506,9.044,148.804
C06127=1149.576,343.901,-78.882,-176.508,9.040,148.804
C06128=1149.580,343.654,-78.848,-176.511,9.036,148.804
C06129=1149.584,343.406,-78.814,-176.514,9.033,148.804
C06130=1149.589,343.159,-78.781,-176.516,9.028,148.803
C06131=1149.592,342.911,-78.746,-176.518,9.025,148.803
C06132=1149.597,342.663,-78.713,-176.521,9.021,148.803
C06133=1149.601,342.416,-78.679,-176.524,9.018,148.803
C06134=1149.605,342.168,-78.646,-176.527,9.014,148.802
C06135=1149.608,341.920,-78.611,-176.529,9.010,148.802
C06136=1149.613,341.672,-78.578,-176.531,9.006,148.802
C06137=1149.617,341.425,-78.544,-176.534,9.003,148.801
C06138=1149.621,341.177,-78.511,-176.537,8.999,148.801
C06139=1149.625,340.929,-78.476,-176.539,8.995,148.801
C06140=1149.629,340.681,-78.443,-176.541,8.991,148.801
C06141=1149.633,340.434,-78.409,-176.544,8.988,148.800
C06142=1149.637,340.187,-78.376,-176.547,8.984,148.800
C06143=1149.640,339.938,-78.342,-176.549,8.980,148.800
C06144=1149.646,339.658,-78.304,-176.552,8.976,148.800
C06145=1149.650,339.378,-78.266,-176.554,8.972,148.799
C06146=1149.655,339.098,-78.228,-176.557,8.968,148.799
C06147=1149.659,338.818,-78.190,-176.560,8.964,148.799
C06148=1149.663,338.571,-78.156,-176.563,8.960,148.798
C06149=1149.668,338.323,-78.122,-176.565,8.956,148.798
C06150=1149.671,338.074,-78.089,-176.568,8.952,148.798
C06151=1149.675,337.826,-78.056,-176.571,8.949,148.798
C06152=1149.679,337.579,-78.022,-176.573,8.945,148.797
C06153=1149.683,337.332,-77.989,-176.575,8.941,148.797
C06154=1149.688,337.084,-77.955,-176.578,8.937,148.797
C06155=1149.692,336.836,-77.922,-176.581,8.934,148.797
C06156=1149.695,336.588,-77.888,-176.584,8.930,148.796
C06157=1149.699,336.341,-77.855,-176.586,8.927,148.796
C06158=1149.703,336.093,-77.822,-176.588,8.923,148.796
C06159=1149.707,335.845,-77.789,-176.591,8.919,148.796
C06160=1149.711,335.597,-77.755,-176.593,8.916,148.795
C06161=1149.716,335.350,-77.722,-176.596,8.912,148.795
C06162=1149.720,335.102,-77.689,-176.598,8.908,148.795
C06163=1149.724,334.855,-77.655,-176.601,8.904,148.795
C06164=1149.727,334.606,-77.622,-176.603,8.901,148.795
C06165=1149.731,334.359,-77.589,-176.606,8.897,148.794
C06166=1149.735,334.111,-77.555,-176.609,8.894,148.794
C06167=1149.740,333.863,-77.522,-176.611,8.890,148.794
C06168=1149.744,333.615,-77.489,-176.614,8.886,148.794
C06169=1149.748,333.368,-77.456,-176.616,8.883,148.793
C06170=1149.752,333.120,-77.423,-176.619,8.879,148.793
C06171=1149.756,332.872,-77.390,-176.621,8.875,148.793
C06172=1149.760,332.625,-77.356,-176.624,8.871,148.793
C06173=1149.764,332.377,-77.323,-176.626,8.868,148.792
C06174=1149.769,332.129,-77.290,-176.629,8.864,148.792
C06175=1149.773,331.881,-77.257,-176.632,8.861,148.792
C06176=1149.777,331.634,-77.224,-176.634,8.857,148.792
C06177=1149.781,331.386,-77.191,-176.637,8.853,148.792
C06178=1149.785,331.138,-77.158,-176.639,8.850,148.791
C06179=1149.789,330.890,-77.126,-176.642,8.846,148.791
C06180=1149.793,330.642,-77.093,-176.644,8.843,148.791
C06181=1149.797,330.395,-77.059,-176.647,8.839,148.791
C06182=1149.801,330.147,-77.026,-176.650,8.835,148.790
C06183=1149.805,329.899,-76.993,-176.652,8.832,148.790
C06184=1149.810,329.651,-76.961,-176.655,8.828,148.790
C06185=1149.813,329.403,-76.928,-176.657,8.825,148.790
C06186=1149.817,329.156,-76.895,-176.660,8.821,148.790
C06187=1149.821,328.908,-76.862,-176.662,8.817,148.789
C06188=1149.826,328.660,-76.829,-176.665,8.814,148.789
C06189=1149.830,328.412,-76.796,-176.668,8.810,148.789
C06190=1149.833,328.164,-76.764,-176.670,8.807,148.789
C06191=1149.838,327.917,-76.730,-176.673,8.803,148.789
C06192=1149.842,327.668,-76.698,-176.675,8.799,148.788
C06193=1149.846,327.421,-76.665,-176.677,8.796,148.788
C06194=1149.850,327.173,-76.632,-176.680,8.792,148.788
C06195=1149.854,326.925,-76.600,-176.683,8.789,148.788
C06196=1149.858,326.677,-76.567,-176.686,8.785,148.787
C06197=1149.863,326.429,-76.534,-176.688,8.781,148.787
C06198=1149.866,326.181,-76.502,-176.690,8.778,148.787
C06199=1149.870,325.934,-76.469,-176.693,8.774,148.787
C06200=1149.875,325.685,-76.436,-176.695,8.771,148.787
C06201=1149.879,325.439,-76.404,-176.698,8.767,148.786
C06202=1149.883,325.190,-76.371,-176.701,8.763,148.786
C06203=1149.887,324.943,-76.338,-176.703,8.760,148.786
C06204=1149.891,324.694,-76.306,-176.706,8.756,148.786
C06205=1149.895,324.447,-76.273,-176.708,8.753,148.786
C06206=1149.899,324.199,-76.241,-176.711,8.749,148.785
C06207=1149.903,323.951,-76.208,-176.713,8.745,148.785
C06208=1149.907,323.703,-76.176,-176.716,8.742,148.785
C06209=1149.911,323.455,-76.143,-176.719,8.738,148.785
C06210=1149.916,323.208,-76.111,-176.721,8.735,148.785
C06211=1149.919,322.960,-76.079,-176.724,8.732,148.785
C06212=1149.924,322.712,-76.046,-176.727,8.728,148.784
C06213=1149.928,322.463,-76.014,-176.729,8.724,148.784
C06214=1149.931,322.216,-75.981,-176.731,8.721,148.784
C06215=1149.936,321.968,-75.949,-176.734,8.717,148.784
C06216=1149.940,321.720,-75.917,-176.737,8.714,148.784
C06217=1149.944,321.473,-75.884,-176.739,8.710,148.783
C06218=1149.948,321.225,-75.852,-176.742,8.706,148.783
C06219=1149.952,320.976,-75.820,-176.744,8.703,148.783
C06220=1149.956,320.729,-75.787,-176.747,8.699,148.783
C06221=1149.960,320.480,-75.755,-176.750,8.696,148.783
C06222=1149.965,320.233,-75.723,-176.752,8.693,148.783
C06223=1149.969,319.985,-75.691,-176.755,8.689,148.782
C06224=1149.972,319.737,-75.658,-176.757,8.685,148.782
C06225=1149.976,319.489,-75.627,-176.760,8.682,148.782
C06226=1149.981,319.242,-75.594,-176.763,8.678,148.782
C06227=1149.985,318.994,-75.563,-176.765,8.675,148.781
C06228=1149.989,318.745,-75.530,-176.768,8.672,148.782
C06229=1149.993,318.498,-75.498,-176.770,8.668,148.781
C06230=1149.998,318.250,-75.466,-176.773,8.664,148.781
C06231=1150.001,318.002,-75.434,-176.775,8.661,148.781
C06232=1150.005,317.754,-75.402,-176.778,8.657,148.781
C06233=1150.010,317.506,-75.369,-176.780,8.654,148.780
C06234=1150.014,317.258,-75.338,-176.783,8.651,148.780
C06235=1150.018,317.010,-75.306,-176.786,8.647,148.780
C06236=1150.022,316.762,-75.274,-176.788,8.644,148.780
C06237=1150.026,316.514,-75.242,-176.791,8.640,148.780
C06238=1150.030,316.267,-75.210,-176.794,8.636,148.780
C06239=1150.035,316.018,-75.178,-176.796,8.633,148.779
C06240=1150.038,315.770,-75.146,-176.799,8.630,148.779
C06241=1150.043,315.523,-75.115,-176.802,8.626,148.779
C06242=1150.047,315.275,-75.082,-176.804,8.623,148.779
C06243=1150.051,315.027,-75.050,-176.806,8.619,148.779
C06244=1150.055,314.779,-75.019,-176.809,8.615,148.779
C06245=1150.059,314.531,-74.986,-176.811,8.612,148.778
C06246=1150.063,314.283,-74.955,-176.814,8.609,148.779
C06247=1150.067,314.036,-74.923,-176.817,8.606,148.778
C06248=1150.072,313.758,-74.887,-176.819,8.602,148.778
C06249=1150.076,313.480,-74.852,-176.822,8.598,148.778
C06250=1150.081,313.203,-74.816,-176.826,8.594,148.778
C06251=1150.086,312.924,-74.781,-176.829,8.590,148.778
C06252=1150.090,312.677,-74.749,-176.831,8.586,148.777
C06253=1150.094,312.429,-74.717,-176.833,8.583,148.777
C06254=1150.098,312.182,-74.686,-176.837,8.579,148.777
C06255=1150.103,311.933,-74.653,-176.839,8.576,148.777
C06256=1150.107,311.685,-74.622,-176.841,8.573,148.777
C06257=1150.111,311.437,-74.591,-176.844,8.569,148.777
C06258=1150.115,311.189,-74.559,-176.847,8.566,148.777
C06259=1150.119,310.941,-74.528,-176.849,8.563,148.776
C06260=1150.123,310.693,-74.496,-176.852,8.559,148.776
C06261=1150.127,310.445,-74.464,-176.854,8.555,148.776
C06262=1150.132,310.198,-74.433,-176.857,8.552,148.776
C06263=1150.136,309.949,-74.401,-176.860,8.549,148.776
C06264=1150.140,309.702,-74.370,-176.862,8.545,148.776
C06265=1150.144,309.454,-74.338,-176.865,8.542,148.775
C06266=1150.148,309.206,-74.307,-176.868,8.539,148.776
C06267=1150.152,308.958,-74.275,-176.870,8.535,148.775
C06268=1150.157,308.710,-74.245,-176.873,8.531,148.775
C06269=1150.160,308.462,-74.213,-176.875,8.528,148.775
C06270=1150.165,308.214,-74.182,-176.878,8.525,148.775
C06271=1150.169,307.966,-74.150,-176.880,8.522,148.775
C06272=1150.173,307.718,-74.119,-176.883,8.518,148.775
C06273=1150.178,307.469,-74.087,-176.886,8.515,148.775
C06274=1150.182,307.222,-74.056,-176.888,8.511,148.774
C06275=1150.186,306.973,-74.024,-176.891,8.507,148.774
C06276=1150.190,306.726,-73.993,-176.894,8.504,148.774
C06277=1150.194,306.477,-73.962,-176.896,8.501,148.774
C06278=1150.199,306.229,-73.931,-176.898,8.498,148.774
C06279=1150.203,305.981,-73.899,-176.902,8.494,148.774
C06280=1150.207,305.734,-73.869,-176.904,8.491,148.774
C06281=1150.210,305.486,-73.837,-176.906,8.488,148.773
C06282=1150.215,305.238,-73.806,-176.909,8.485,148.773
C06283=1150.219,304.990,-73.775,-176.912,8.481,148.773
C06284=1150.223,304.742,-73.744,-176.914,8.477,148.773
C06285=1150.228,304.494,-73.713,-176.917,8.474,148.773
C06286=1150.231,304.246,-73.681,-176.920,8.471,148.773
C06287=1150.236,303.998,-73.650,-176.922,8.467,148.773
C06288=1150.240,303.749,-73.619,-176.925,8.464,148.773
C06289=1150.244,303.502,-73.588,-176.927,8.461,148.773
C06290=1150.248,303.253,-73.557,-176.930,8.457,148.772
C06291=1150.253,303.005,-73.526,-176.933,8.454,148.772
C06292=1150.257,302.758,-73.496,-176.935,8.450,148.772
C06293=1150.261,302.509,-73.464,-176.938,8.447,148.772
C06294=1150.265,302.262,-73.433,-176.941,8.444,148.772
C06295=1150.269,302.013,-73.402,-176.943,8.440,148.772
C06296=1150.274,301.765,-73.371,-176.946,8.437,148.772
C06297=1150.278,301.517,-73.340,-176.949,8.434,148.772
C06298=1150.281,301.269,-73.309,-176.951,8.431,148.772
C06299=1150.286,301.021,-73.278,-176.954,8.428,148.772
C06300=1150.291,300.773,-73.248,-176.957,8.424,148.771
C06301=1150.295,300.525,-73.217,-176.959,8.421,148.771
C06302=1150.299,300.277,-73.186,-176.962,8.417,148.771
C06303=1150.303,300.029,-73.156,-176.964,8.414,148.771
C06304=1150.307,299.780,-73.125,-176.967,8.410,148.771
C06305=1150.312,299.532,-73.094,-176.970,8.407,148.771
C06306=1150.316,299.284,-73.063,-176.972,8.404,148.771
C06307=1150.320,299.036,-73.032,-176.975,8.401,148.771
C06308=1150.324,298.788,-73.002,-176.977,8.398,148.771
C06309=1150.329,298.540,-72.971,-176.980,8.394,148.770
C06310=1150.332,298.292,-72.940,-176.983,8.391,148.770
C06311=1150.337,298.044,-72.910,-176.985,8.388,148.770
C06312=1150.341,297.796,-72.879,-176.988,8.384,148.770
C06313=1150.345,297.548,-72.848,-176.991,8.381,148.770
C06314=1150.349,297.300,-72.818,-176.993,8.377,148.770
C06315=1150.354,297.052,-72.787,-176.996,8.374,148.770
C06316=1150.358,296.804,-72.757,-176.999,8.371,148.770
C06317=1150.362,296.555,-72.726,-177.001,8.368,148.770
C06318=1150.366,296.307,-72.695,-177.004,8.364,148.770
C06319=1150.370,296.060,-72.665,-177.007,8.361,148.770
C06320=1150.375,295.812,-72.634,-177.009,8.358,148.770
C06321=1150.378,295.563,-72.603,-177.012,8.355,148.769
C06322=1150.383,295.315,-72.573,-177.014,8.352,148.769
C06323=1150.388,295.067,-72.542,-177.017,8.347,148.769
C06324=1150.392,294.819,-72.512,-177.020,8.345,148.769
C06325=1150.396,294.571,-72.481,-177.022,8.341,148.769
C06326=1150.399,294.323,-72.451,-177.025,8.338,148.769
C06327=1150.404,294.074,-72.421,-177.027,8.335,148.769
C06328=1150.408,293.827,-72.391,-177.030,8.332,148.769
C06329=1150.413,293.579,-72.360,-177.033,8.328,148.769
C06330=1150.416,293.330,-72.329,-177.036,8.325,148.769
C06331=1150.421,293.082,-72.299,-177.038,8.322,148.769
C06332=1150.425,292.834,-72.269,-177.041,8.319,148.769
C06333=1150.430,292.586,-72.238,-177.043,8.316,148.768
C06334=1150.434,292.338,-72.209,-177.047,8.312,148.768
C06335=1150.438,292.089,-72.178,-177.049,8.309,148.768
C06336=1150.442,291.842,-72.148,-177.052,8.306,148.768
C06337=1150.447,291.593,-72.118,-177.054,8.302,148.768
C06338=1150.450,291.345,-72.088,-177.057,8.299,148.768
C06339=1150.454,291.098,-72.057,-177.060,8.296,148.768
C06340=1150.459,290.849,-72.027,-177.063,8.292,148.768
C06341=1150.463,290.601,-71.997,-177.065,8.289,148.768
C06342=1150.467,290.352,-71.967,-177.068,8.286,148.768
C06343=1150.471,290.105,-71.937,-177.070,8.283,148.768
C06344=1150.476,289.856,-71.907,-177.073,8.280,148.768
C06345=1150.480,289.608,-71.876,-177.075,8.277,148.768
C06346=1150.484,289.360,-71.847,-177.078,8.274,148.768
C06347=1150.489,289.112,-71.816,-177.081,8.270,148.768
C06348=1150.493,288.864,-71.787,-177.083,8.267,148.767
C06349=1150.497,288.616,-71.757,-177.086,8.264,148.767
C06350=1150.501,288.367,-71.726,-177.089,8.261,148.768
C06351=1150.505,288.119,-71.696,-177.091,8.258,148.767
C06352=1150.510,287.844,-71.663,-177.095,8.254,148.767
C06353=1150.515,287.569,-71.630,-177.097,8.250,148.767
C06354=1150.519,287.293,-71.597,-177.100,8.247,148.767
C06355=1150.524,287.018,-71.563,-177.104,8.243,148.767
C06356=1150.529,286.770,-71.534,-177.106,8.240,148.767
C06357=1150.533,286.522,-71.503,-177.109,8.237,148.767
C06358=1150.537,286.274,-71.474,-177.112,8.234,148.767
C06359=1150.542,286.025,-71.444,-177.114,8.231,148.767
C06360=1150.545,285.778,-71.414,-177.117,8.228,148.767
C06361=1150.550,285.529,-71.384,-177.119,8.224,148.767
C06362=1150.554,285.281,-71.355,-177.122,8.221,148.767
C06363=1150.559,285.032,-71.325,-177.125,8.218,148.767
C06364=1150.563,284.785,-71.295,-177.127,8.214,148.767
C06365=1150.567,284.537,-71.265,-177.130,8.211,148.767
C06366=1150.571,284.288,-71.236,-177.133,8.208,148.767
C06367=1150.575,284.040,-71.206,-177.135,8.205,148.767
C06368=1150.580,283.792,-71.176,-177.138,8.202,148.767
C06369=1150.584,283.544,-71.146,-177.140,8.199,148.766
C06370=1150.588,283.296,-71.117,-177.144,8.195,148.766
C06371=1150.592,283.047,-71.087,-177.147,8.192,148.767
C06372=1150.597,282.799,-71.058,-177.149,8.189,148.766
C06373=1150.601,282.551,-71.028,-177.152,8.186,148.766
C06374=1150.606,282.302,-70.998,-177.154,8.183,148.766
C06375=1150.610,282.054,-70.969,-177.157,8.180,148.766
C06376=1150.614,281.806,-70.939,-177.159,8.177,148.766
C06377=1150.618,281.558,-70.909,-177.162,8.174,148.766
C06378=1150.622,281.310,-70.880,-177.165,8.170,148.766
C06379=1150.626,281.061,-70.850,-177.168,8.167,148.766
C06380=1150.631,280.814,-70.821,-177.170,8.164,148.766
C06381=1150.635,280.566,-70.792,-177.173,8.161,148.766
C06382=1150.639,280.317,-70.762,-177.176,8.158,148.766
C06383=1150.644,280.069,-70.733,-177.178,8.155,148.766
C06384=1150.648,279.821,-70.703,-177.181,8.152,148.766
C06385=1150.652,279.573,-70.674,-177.184,8.149,148.766
C06386=1150.656,279.324,-70.644,-177.186,8.146,148.766
C06387=1150.660,279.076,-70.615,-177.189,8.142,148.766
C06388=1150.665,278.827,-70.586,-177.192,8.139,148.766
C06389=1150.669,278.579,-70.557,-177.195,8.136,148.766
C06390=1150.674,278.331,-70.528,-177.197,8.132,148.766
C06391=1150.678,278.083,-70.498,-177.200,8.129,148.766
C06392=1150.682,277.835,-70.469,-177.203,8.127,148.766
C06393=1150.686,277.586,-70.439,-177.205,8.123,148.766
C06394=1150.690,277.338,-70.410,-177.208,8.120,148.766
C06395=1150.695,277.089,-70.381,-177.211,8.117,148.766
C06396=1150.699,276.841,-70.352,-177.213,8.114,148.766
C06397=1150.704,276.594,-70.323,-177.216,8.111,148.766
C06398=1150.708,276.345,-70.293,-177.218,8.108,148.766
C06399=1150.712,276.097,-70.264,-177.221,8.105,148.766
C06400=1150.717,275.848,-70.235,-177.224,8.102,148.766
C06401=1150.720,275.600,-70.206,-177.227,8.098,148.766
C06402=1150.724,275.352,-70.177,-177.230,8.095,148.766
C06403=1150.729,275.104,-70.148,-177.232,8.092,148.766
C06404=1150.734,274.855,-70.119,-177.235,8.089,148.766
C06405=1150.738,274.607,-70.089,-177.238,8.086,148.766
C06406=1150.742,274.359,-70.060,-177.240,8.083,148.766
C06407=1150.746,274.110,-70.032,-177.243,8.080,148.766
C06408=1150.751,273.863,-70.003,-177.245,8.077,148.766
C06409=1150.755,273.614,-69.973,-177.248,8.074,148.766
C06410=1150.759,273.366,-69.945,-177.251,8.071,148.766
C06411=1150.763,273.117,-69.915,-177.254,8.068,148.766
C06412=1150.768,272.869,-69.887,-177.256,8.065,148.766
C06413=1150.772,272.621,-69.858,-177.259,8.062,148.766
C06414=1150.776,272.372,-69.829,-177.262,8.059,148.766
C06415=1150.781,272.124,-69.800,-177.264,8.056,148.766
C06416=1150.785,271.876,-69.771,-177.267,8.053,148.766
C06417=1150.789,271.628,-69.742,-177.269,8.050,148.766
C06418=1150.793,271.380,-69.713,-177.273,8.046,148.766
C06419=1150.798,271.131,-69.685,-177.276,8.043,148.766
C06420=1150.802,270.883,-69.656,-177.278,8.040,148.766
C06421=1150.806,270.635,-69.627,-177.281,8.037,148.766
C06422=1150.811,270.386,-69.598,-177.283,8.034,148.766
C06423=1150.816,270.138,-69.569,-177.286,8.031,148.766
C06424=1150.819,269.890,-69.541,-177.289,8.028,148.766
C06425=1150.824,269.641,-69.512,-177.292,8.025,148.766
C06426=1150.829,269.393,-69.483,-177.295,8.022,148.766
C06427=1150.832,269.145,-69.455,-177.297,8.019,148.766
C06428=1150.837,268.896,-69.426,-177.300,8.016,148.766
C06429=1150.842,268.648,-69.397,-177.302,8.013,148.766
C06430=1150.845,268.400,-69.368,-177.305,8.010,148.766
C06431=1150.850,268.151,-69.340,-177.308,8.007,148.766
C06432=1150.854,267.903,-69.312,-177.310,8.004,148.766
C06433=1150.858,267.654,-69.283,-177.313,8.001,148.766
C06434=1150.863,267.407,-69.254,-177.316,7.998,148.766
C06435=1150.867,267.158,-69.226,-177.319,7.995,148.766
C06436=1150.871,266.909,-69.197,-177.321,7.992,148.766
C06437=1150.875,266.662,-69.169,-177.324,7.989,148.766
C06438=1150.880,266.413,-69.140,-177.327,7.986,148.766
C06439=1150.884,266.165,-69.112,-177.329,7.983,148.766
C06440=1150.889,265.917,-69.083,-177.332,7.980,148.766
C06441=1150.893,265.668,-69.055,-177.335,7.977,148.766
C06442=1150.897,265.420,-69.026,-177.338,7.974,148.766
C06443=1150.902,265.171,-68.997,-177.340,7.971,148.766
C06444=1150.906,264.924,-68.970,-177.343,7.968,148.766
C06445=1150.911,264.675,-68.941,-177.346,7.965,148.766
C06446=1150.914,264.426,-68.913,-177.348,7.962,148.766
C06447=1150.920,264.178,-68.884,-177.351,7.959,148.766
C06448=1150.923,263.929,-68.856,-177.354,7.956,148.766
C06449=1150.928,263.681,-68.828,-177.357,7.953,148.766
C06450=1150.932,263.433,-68.800,-177.359,7.950,148.766
C06451=1150.936,263.185,-68.771,-177.362,7.948,148.767
C06452=1150.941,262.936,-68.743,-177.365,7.945,148.767
C06453=1150.945,262.689,-68.715,-177.367,7.941,148.766
C06454=1150.949,262.440,-68.686,-177.370,7.938,148.766
C06455=1150.954,262.192,-68.658,-177.373,7.935,148.767
C06456=1150.958,261.918,-68.627,-177.376,7.932,148.767
C06457=1150.963,261.644,-68.596,-177.379,7.929,148.767
C06458=1150.968,261.371,-68.565,-177.382,7.926,148.767
C06459=1150.973,261.097,-68.535,-177.385,7.922,148.767
C06460=1150.978,260.849,-68.506,-177.388,7.919,148.767
C06461=1150.981,260.601,-68.478,-177.391,7.916,148.767
C06462=1150.986,260.353,-68.450,-177.393,7.913,148.767
C06463=1150.990,260.104,-68.422,-177.396,7.910,148.767
C06464=1150.995,259.856,-68.394,-177.399,7.907,148.767
C06465=1150.998,259.608,-68.366,-177.402,7.904,148.767
C06466=1151.003,259.359,-68.337,-177.405,7.902,148.767
C06467=1151.008,259.110,-68.310,-177.407,7.898,148.767
C06468=1151.012,258.862,-68.282,-177.409,7.896,148.767
C06469=1151.016,258.614,-68.254,-177.412,7.893,148.767
C06470=1151.021,258.365,-68.226,-177.415,7.890,148.767
C06471=1151.025,258.118,-68.198,-177.417,7.887,148.767
C06472=1151.029,257.868,-68.170,-177.420,7.884,148.767
C06473=1151.034,257.620,-68.142,-177.423,7.881,148.767
C06474=1151.038,257.372,-68.114,-177.426,7.879,148.767
C06475=1151.042,257.124,-68.086,-177.429,7.876,148.768
C06476=1151.047,256.875,-68.059,-177.431,7.873,148.768
C06477=1151.051,256.627,-68.031,-177.434,7.870,148.768
C06478=1151.056,256.379,-68.002,-177.437,7.867,148.768
C06479=1151.060,256.129,-67.975,-177.440,7.864,148.768
C06480=1151.064,255.881,-67.947,-177.442,7.861,148.768
C06481=1151.069,255.634,-67.919,-177.445,7.858,148.768
C06482=1151.073,255.384,-67.892,-177.448,7.855,148.768
C06483=1151.078,255.136,-67.864,-177.451,7.852,148.768
C06484=1151.082,254.888,-67.837,-177.454,7.849,148.768
C06485=1151.086,254.639,-67.808,-177.456,7.846,148.768
C06486=1151.090,254.391,-67.781,-177.459,7.843,148.768
C06487=1151.095,254.143,-67.754,-177.462,7.840,148.768
C06488=1151.099,253.894,-67.725,-177.465,7.837,148.768
C06489=1151.104,253.646,-67.698,-177.467,7.835,148.768
C06490=1151.108,253.398,-67.671,-177.469,7.832,148.768
C06491=1151.113,253.148,-67.643,-177.472,7.829,148.768
C06492=1151.117,252.900,-67.615,-177.475,7.826,148.768
C06493=1151.122,252.652,-67.588,-177.477,7.823,148.769
C06494=1151.125,252.403,-67.560,-177.480,7.820,148.769
C06495=1151.130,252.155,-67.533,-177.483,7.817,148.769
C06496=1151.134,251.907,-67.505,-177.486,7.814,148.769
C06497=1151.138,251.658,-67.477,-177.489,7.811,148.769
C06498=1151.143,251.409,-67.450,-177.491,7.809,148.769
C06499=1151.147,251.161,-67.423,-177.495,7.806,148.769
C06500=1151.152,250.913,-67.395,-177.497,7.803,148.769
C06501=1151.156,250.664,-67.367,-177.500,7.800,148.769
C06502=1151.161,250.416,-67.340,-177.502,7.798,148.769
C06503=1151.165,250.167,-67.313,-177.505,7.795,148.769
C06504=1151.169,249.919,-67.285,-177.508,7.792,148.770
C06505=1151.174,249.670,-67.258,-177.511,7.789,148.770
C06506=1151.178,249.422,-67.231,-177.514,7.786,148.770
C06507=1151.183,249.174,-67.203,-177.516,7.783,148.770
C06508=1151.187,248.925,-67.176,-177.519,7.780,148.770
C06509=1151.191,248.676,-67.149,-177.522,7.777,148.770
C06510=1151.196,248.428,-67.122,-177.525,7.775,148.770
C06511=1151.200,248.180,-67.094,-177.527,7.772,148.770
C06512=1151.204,247.932,-67.067,-177.530,7.769,148.770
C06513=1151.208,247.682,-67.040,-177.532,7.767,148.770
C06514=1151.213,247.434,-67.013,-177.535,7.764,148.770
C06515=1151.217,247.186,-66.985,-177.538,7.761,148.770
C06516=1151.222,246.938,-66.958,-177.541,7.758,148.770
C06517=1151.227,246.689,-66.931,-177.544,7.755,148.770
C06518=1151.231,246.440,-66.904,-177.546,7.752,148.771
C06519=1151.235,246.191,-66.877,-177.549,7.749,148.771
C06520=1151.239,245.943,-66.850,-177.552,7.746,148.771
C06521=1151.244,245.695,-66.823,-177.555,7.743,148.771
C06522=1151.249,245.446,-66.796,-177.557,7.741,148.771
C06523=1151.253,245.198,-66.768,-177.560,7.738,148.771
C06524=1151.258,244.950,-66.741,-177.563,7.735,148.771
C06525=1151.261,244.701,-66.714,-177.566,7.732,148.771
C06526=1151.266,244.452,-66.687,-177.568,7.730,148.771
C06527=1151.270,244.204,-66.660,-177.571,7.727,148.771
C06528=1151.275,243.955,-66.633,-177.574,7.724,148.772
C06529=1151.279,243.707,-66.607,-177.577,7.721,148.772
C06530=1151.283,243.459,-66.580,-177.579,7.719,148.772
C06531=1151.288,243.210,-66.552,-177.582,7.716,148.772
C06532=1151.292,242.961,-66.525,-177.585,7.713,148.772
C06533=1151.296,242.713,-66.499,-177.587,7.710,148.772
C06534=1151.301,242.464,-66.472,-177.591,7.707,148.772
C06535=1151.305,242.216,-66.444,-177.593,7.704,148.772
C06536=1151.310,241.967,-66.418,-177.596,7.701,148.772
C06537=1151.314,241.719,-66.392,-177.598,7.699,148.772
C06538=1151.319,241.470,-66.365,-177.601,7.696,148.773
C06539=1151.324,241.222,-66.338,-177.604,7.693,148.773
C06540=1151.328,240.973,-66.311,-177.607,7.690,148.773
C06541=1151.332,240.725,-66.284,-177.609,7.688,148.773
C06542=1151.337,240.476,-66.257,-177.612,7.685,148.773
C06543=1151.341,240.228,-66.231,-177.615,7.683,148.773
C06544=1151.346,239.979,-66.204,-177.618,7.680,148.773
C06545=1151.350,239.731,-66.178,-177.620,7.677,148.773
C06546=1151.354,239.482,-66.151,-177.623,7.674,148.773
C06547=1151.359,239.234,-66.124,-177.626,7.671,148.773
C06548=1151.363,238.985,-66.098,-177.629,7.668,148.774
C06549=1151.368,238.737,-66.071,-177.632,7.665,148.774
C06550=1151.372,238.489,-66.044,-177.634,7.663,148.774
C06551=1151.377,238.239,-66.018,-177.637,7.661,148.774
C06552=1151.381,237.991,-65.991,-177.640,7.658,148.774
C06553=1151.385,237.743,-65.964,-177.643,7.655,148.774
C06554=1151.390,237.494,-65.937,-177.645,7.652,148.774
C06555=1151.394,237.245,-65.912,-177.648,7.650,148.774
C06556=1151.399,236.997,-65.885,-177.650,7.647,148.774
C06557=1151.403,236.748,-65.859,-177.653,7.644,148.775
C06558=1151.408,236.500,-65.832,-177.656,7.641,148.775
C06559=1151.412,236.251,-65.805,-177.659,7.638,148.775
C06560=1151.417,235.979,-65.777,-177.662,7.635,148.775
C06561=1151.422,235.707,-65.747,-177.665,7.632,148.775
C06562=1151.426,235.436,-65.718,-177.668,7.630,148.775
C06563=1151.431,235.163,-65.689,-177.671,7.627,148.775
C06564=1151.435,234.915,-65.663,-177.674,7.624,148.776
C06565=1151.440,234.666,-65.637,-177.676,7.621,148.776
C06566=1151.444,234.418,-65.610,-177.679,7.618,148.776
C06567=1151.448,234.169,-65.584,-177.682,7.616,148.776
C06568=1151.454,233.921,-65.558,-177.685,7.613,148.776
C06569=1151.458,233.673,-65.532,-177.687,7.611,148.776
C06570=1151.463,233.424,-65.505,-177.690,7.608,148.776
C06571=1151.467,233.175,-65.479,-177.693,7.605,148.776
C06572=1151.471,232.927,-65.453,-177.696,7.602,148.777
C06573=1151.476,232.678,-65.426,-177.698,7.600,148.777
C06574=1151.480,232.429,-65.401,-177.701,7.597,148.777
C06575=1151.485,232.181,-65.374,-177.704,7.594,148.777
C06576=1151.489,231.932,-65.348,-177.707,7.591,148.777
C06577=1151.493,231.684,-65.322,-177.710,7.589,148.777
C06578=1151.498,231.435,-65.295,-177.712,7.586,148.777
C06579=1151.502,231.186,-65.270,-177.715,7.584,148.778
C06580=1151.506,230.938,-65.243,-177.718,7.581,148.778
C06581=1151.511,230.689,-65.217,-177.721,7.578,148.778
C06582=1151.516,230.440,-65.191,-177.723,7.576,148.778
C06583=1151.520,230.192,-65.166,-177.726,7.573,148.778
C06584=1151.524,229.944,-65.139,-177.729,7.570,148.778
C06585=1151.529,229.695,-65.113,-177.732,7.567,148.778
C06586=1151.534,229.446,-65.087,-177.735,7.565,148.779
C06587=1151.537,229.198,-65.061,-177.737,7.562,148.779
C06588=1151.542,228.949,-65.035,-177.740,7.560,148.779
C06589=1151.547,228.701,-65.009,-177.743,7.557,148.779
C06590=1151.551,228.452,-64.983,-177.745,7.554,148.779
C06591=1151.556,228.203,-64.957,-177.748,7.552,148.779
C06592=1151.560,227.955,-64.931,-177.751,7.549,148.779
C06593=1151.565,227.706,-64.905,-177.754,7.546,148.779
C06594=1151.569,227.458,-64.879,-177.756,7.543,148.780
C06595=1151.574,227.209,-64.853,-177.759,7.541,148.780
C06596=1151.578,226.960,-64.828,-177.762,7.538,148.780
C06597=1151.582,226.711,-64.802,-177.765,7.535,148.780
C06598=1151.588,226.463,-64.776,-177.767,7.533,148.780
C06599=1151.592,226.214,-64.750,-177.770,7.531,148.780
C06600=1151.596,225.965,-64.724,-177.773,7.528,148.781
C06601=1151.600,225.716,-64.699,-177.776,7.525,148.781
C06602=1151.605,225.469,-64.673,-177.779,7.522,148.781
C06603=1151.609,225.220,-64.647,-177.781,7.520,148.781
C06604=1151.613,224.971,-64.621,-177.784,7.517,148.781
C06605=1151.618,224.723,-64.596,-177.787,7.514,148.781
C06606=1151.623,224.474,-64.569,-177.789,7.513,148.782
C06607=1151.627,224.225,-64.544,-177.792,7.510,148.782
C06608=1151.632,223.976,-64.519,-177.795,7.507,148.782
C06609=1151.637,223.728,-64.493,-177.798,7.504,148.782
C06610=1151.641,223.479,-64.467,-177.800,7.502,148.782
C06611=1151.645,223.230,-64.442,-177.803,7.499,148.782
C06612=1151.650,222.982,-64.416,-177.806,7.496,148.782
C06613=1151.654,222.733,-64.391,-177.809,7.493,148.782
C06614=1151.658,222.484,-64.365,-177.812,7.492,148.783
C06615=1151.663,222.236,-64.339,-177.814,7.489,148.783
C06616=1151.667,221.988,-64.314,-177.817,7.486,148.783
C06617=1151.672,221.739,-64.288,-177.820,7.484,148.783
C06618=1151.677,221.490,-64.263,-177.823,7.481,148.783
C06619=1151.681,221.241,-64.238,-177.825,7.478,148.783
C06620=1151.686,220.993,-64.212,-177.828,7.476,148.784
C06621=1151.690,220.744,-64.186,-177.831,7.473,148.784
C06622=1151.694,220.496,-64.161,-177.834,7.470,148.784
C06623=1151.699,220.247,-64.136,-177.837,7.468,148.784
C06624=1151.704,219.998,-64.110,-177.839,7.466,148.784
C06625=1151.708,219.749,-64.084,-177.842,7.463,148.784
C06626=1151.713,219.501,-64.059,-177.845,7.460,148.785
C06627=1151.717,219.252,-64.034,-177.847,7.458,148.785
C06628=1151.722,219.004,-64.009,-177.850,7.455,148.785
C06629=1151.726,218.755,-63.984,-177.853,7.452,148.785
C06630=1151.730,218.506,-63.958,-177.856,7.451,148.785
C06631=1151.735,218.258,-63.933,-177.858,7.448,148.786
C06632=1151.739,218.009,-63.907,-177.861,7.445,148.786
C06633=1151.744,217.760,-63.883,-177.864,7.443,148.786
C06634=1151.748,217.511,-63.857,-177.867,7.440,148.786
C06635=1151.753,217.263,-63.832,-177.869,7.437,148.786
C06636=1151.757,217.014,-63.807,-177.872,7.435,148.786
C06637=1151.761,216.765,-63.781,-177.875,7.432,148.787
C06638=1151.766,216.516,-63.757,-177.878,7.430,148.787
C06639=1151.771,216.268,-63.731,-177.880,7.428,148.787
C06640=1151.775,216.020,-63.706,-177.883,7.425,148.787
C06641=1151.779,215.770,-63.681,-177.886,7.422,148.787
C06642=1151.784,215.522,-63.656,-177.889,7.420,148.788
C06643=1151.789,215.273,-63.631,-177.891,7.417,148.788
C06644=1151.793,215.025,-63.605,-177.895,7.415,148.788
C06645=1151.798,214.775,-63.580,-177.897,7.413,148.788
C06646=1151.802,214.528,-63.555,-177.900,7.410,148.788
C06647=1151.807,214.278,-63.530,-177.903,7.407,148.788
C06648=1151.811,214.030,-63.505,-177.905,7.405,148.789
C06649=1151.816,213.781,-63.480,-177.908,7.402,148.789
C06650=1151.820,213.532,-63.456,-177.911,7.399,148.789
C06651=1151.825,213.283,-63.430,-177.913,7.397,148.789
C06652=1151.830,213.035,-63.406,-177.917,7.395,148.789
C06653=1151.833,212.786,-63.380,-177.919,7.393,148.790
C06654=1151.838,212.537,-63.356,-177.922,7.390,148.790
C06655=1151.843,212.288,-63.331,-177.925,7.387,148.790
C06656=1151.847,212.040,-63.306,-177.927,7.385,148.790
C06657=1151.852,211.792,-63.281,-177.930,7.382,148.790
C06658=1151.857,211.542,-63.256,-177.933,7.380,148.791
C06659=1151.861,211.294,-63.231,-177.935,7.377,148.791
C06660=1151.865,211.045,-63.206,-177.939,7.375,148.791
C06661=1151.870,210.796,-63.182,-177.941,7.373,148.791
C06662=1151.874,210.548,-63.157,-177.944,7.370,148.791
C06663=1151.879,210.299,-63.132,-177.947,7.367,148.792
C06664=1151.884,210.029,-63.105,-177.950,7.364,148.792
C06665=1151.889,209.758,-63.078,-177.953,7.362,148.792
C06666=1151.894,209.488,-63.051,-177.955,7.360,148.792
C06667=1151.898,209.217,-63.024,-177.958,7.357,148.792
C06668=1151.904,208.968,-63.000,-177.961,7.354,148.792
C06669=1151.907,208.719,-62.975,-177.964,7.352,148.793
C06670=1151.912,208.470,-62.950,-177.967,7.349,148.793
C06671=1151.918,208.222,-62.926,-177.970,7.347,148.793
C06672=1151.921,207.972,-62.901,-177.972,7.345,148.793
C06673=1151.926,207.724,-62.876,-177.975,7.342,148.794
C06674=1151.931,207.476,-62.852,-177.978,7.339,148.794
C06675=1151.935,207.227,-62.827,-177.980,7.337,148.794
C06676=1151.940,206.978,-62.803,-177.984,7.335,148.794
C06677=1151.945,206.729,-62.778,-177.986,7.333,148.794
C06678=1151.948,206.480,-62.754,-177.989,7.330,148.795
C06679=1151.954,206.232,-62.729,-177.992,7.327,148.795
C06680=1151.958,205.983,-62.705,-177.995,7.325,148.795
C06681=1151.963,205.734,-62.680,-177.997,7.322,148.795
C06682=1151.967,205.485,-62.656,-178.000,7.321,148.796
C06683=1151.972,205.237,-62.631,-178.003,7.318,148.796
C06684=1151.976,204.987,-62.607,-178.005,7.316,148.796
C06685=1151.980,204.739,-62.583,-178.008,7.313,148.796
C06686=1151.985,204.490,-62.558,-178.011,7.310,148.796
C06687=1151.990,204.242,-62.534,-178.014,7.308,148.797
C06688=1151.994,203.992,-62.509,-178.017,7.305,148.797
C06689=1151.999,203.744,-62.485,-178.019,7.304,148.797
C06690=1152.003,203.496,-62.461,-178.022,7.301,148.797
C06691=1152.008,203.247,-62.436,-178.025,7.299,148.797
C06692=1152.012,202.998,-62.412,-178.028,7.296,148.798
C06693=1152.017,202.749,-62.387,-178.030,7.294,148.798
C06694=1152.022,202.500,-62.364,-178.033,7.291,148.798
C06695=1152.026,202.252,-62.340,-178.036,7.289,148.798
C06696=1152.031,202.002,-62.314,-178.039,7.287,148.798
C06697=1152.035,201.754,-62.290,-178.042,7.284,148.799
C06698=1152.040,201.505,-62.266,-178.044,7.282,148.799
C06699=1152.045,201.257,-62.242,-178.047,7.279,148.799
C06700=1152.049,201.007,-62.218,-178.049,7.277,148.799
C06701=1152.053,200.759,-62.194,-178.053,7.275,148.800
C06702=1152.058,200.510,-62.170,-178.055,7.273,148.800
C06703=1152.063,200.261,-62.145,-178.058,7.270,148.800
C06704=1152.067,200.012,-62.122,-178.060,7.268,148.800
C06705=1152.071,199.763,-62.097,-178.064,7.265,148.801
C06706=1152.076,199.515,-62.073,-178.066,7.263,148.801
C06707=1152.081,199.266,-62.049,-178.069,7.261,148.801
C06708=1152.085,199.017,-62.025,-178.072,7.258,148.801
C06709=1152.090,198.769,-62.001,-178.075,7.256,148.802
C06710=1152.094,198.520,-61.977,-178.077,7.253,148.802
C06711=1152.099,198.270,-61.953,-178.080,7.251,148.802
C06712=1152.103,198.022,-61.929,-178.083,7.249,148.802
C06713=1152.108,197.773,-61.905,-178.086,7.247,148.802
C06714=1152.113,197.524,-61.881,-178.088,7.244,148.803
C06715=1152.117,197.276,-61.857,-178.091,7.242,148.803
C06716=1152.122,197.027,-61.833,-178.094,7.239,148.803
C06717=1152.126,196.777,-61.809,-178.097,7.237,148.803
C06718=1152.131,196.529,-61.785,-178.099,7.235,148.803
C06719=1152.135,196.280,-61.761,-178.102,7.233,148.804
C06720=1152.140,196.032,-61.737,-178.105,7.230,148.804
C06721=1152.144,195.783,-61.714,-178.108,7.228,148.804
C06722=1152.149,195.534,-61.690,-178.111,7.226,148.805
C06723=1152.154,195.285,-61.666,-178.113,7.223,148.805
C06724=1152.159,195.036,-61.642,-178.116,7.221,148.805
C06725=1152.163,194.787,-61.618,-178.118,7.219,148.805
C06726=1152.168,194.539,-61.594,-178.122,7.216,148.806
C06727=1152.172,194.289,-61.571,-178.124,7.214,148.806
C06728=1152.176,194.041,-61.547,-178.127,7.212,148.806
C06729=1152.181,193.792,-61.523,-178.129,7.209,148.806
C06730=1152.186,193.543,-61.500,-178.133,7.207,148.806
C06731=1152.190,193.294,-61.476,-178.135,7.205,148.807
C06732=1152.195,193.045,-61.452,-178.138,7.202,148.807
C06733=1152.199,192.797,-61.428,-178.141,7.200,148.807
C06734=1152.204,192.548,-61.405,-178.144,7.198,148.807
C06735=1152.208,192.299,-61.382,-178.146,7.196,148.808
C06736=1152.213,192.050,-61.358,-178.149,7.193,148.808
C06737=1152.218,191.801,-61.334,-178.152,7.191,148.808
C06738=1152.222,191.552,-61.311,-178.155,7.189,148.809
C06739=1152.227,191.304,-61.287,-178.157,7.186,148.809
C06740=1152.231,191.055,-61.263,-178.161,7.184,148.809
C06741=1152.236,190.806,-61.240,-178.163,7.182,148.809
C06742=1152.240,190.557,-61.216,-178.166,7.180,148.810
C06743=1152.245,190.308,-61.193,-178.169,7.178,148.810
C06744=1152.250,190.059,-61.169,-178.171,7.175,148.810
C06745=1152.255,189.810,-61.146,-178.174,7.173,148.810
C06746=1152.259,189.562,-61.122,-178.176,7.171,148.810
C06747=1152.264,189.313,-61.098,-178.180,7.168,148.811
C06748=1152.268,189.064,-61.075,-178.182,7.166,148.811
C06749=1152.273,188.815,-61.052,-178.185,7.164,148.811
C06750=1152.278,188.566,-61.028,-178.188,7.162,148.812
C06751=1152.282,188.317,-61.005,-178.191,7.159,148.812
C06752=1152.287,188.068,-60.981,-178.193,7.157,148.812
C06753=1152.291,187.820,-60.958,-178.196,7.155,148.812
C06754=1152.296,187.571,-60.935,-178.199,7.152,148.813
C06755=1152.301,187.322,-60.912,-178.202,7.151,148.813
C06756=1152.305,187.073,-60.888,-178.204,7.148,148.813
C06757=1152.310,186.824,-60.865,-178.207,7.146,148.813
C06758=1152.315,186.575,-60.842,-178.210,7.143,148.814
C06759=1152.319,186.326,-60.819,-178.213,7.141,148.814
C06760=1152.324,186.077,-60.796,-178.215,7.140,148.814
C06761=1152.328,185.828,-60.772,-178.219,7.137,148.815
C06762=1152.333,185.579,-60.749,-178.221,7.135,148.815
C06763=1152.338,185.330,-60.726,-178.224,7.132,148.815
C06764=1152.342,185.082,-60.703,-178.227,7.131,148.815
C06765=1152.347,184.833,-60.680,-178.230,7.128,148.816
C06766=1152.352,184.584,-60.656,-178.232,7.126,148.816
C06767=1152.356,184.335,-60.633,-178.234,7.124,148.816
C06768=1152.361,184.066,-60.608,-178.238,7.121,148.816
C06769=1152.366,183.797,-60.583,-178.241,7.119,148.817
C06770=1152.371,183.527,-60.558,-178.244,7.116,148.817
C06771=1152.376,183.256,-60.532,-178.247,7.115,148.817
C06772=1152.380,183.008,-60.510,-178.250,7.112,148.818
C06773=1152.385,182.759,-60.487,-178.252,7.110,148.818
C06774=1152.390,182.510,-60.463,-178.255,7.108,148.818
C06775=1152.394,182.262,-60.441,-178.258,7.105,148.818
C06776=1152.399,182.013,-60.417,-178.261,7.103,148.819
C06777=1152.404,181.763,-60.395,-178.264,7.101,148.819
C06778=1152.408,181.515,-60.372,-178.266,7.099,148.819
C06779=1152.413,181.266,-60.349,-178.269,7.097,148.820
C06780=1152.417,181.017,-60.325,-178.272,7.095,148.820
C06781=1152.421,180.768,-60.303,-178.274,7.092,148.820
C06782=1152.426,180.518,-60.280,-178.278,7.090,148.820
C06783=1152.432,180.270,-60.257,-178.280,7.088,148.821
C06784=1152.436,180.021,-60.234,-178.282,7.086,148.821
C06785=1152.440,179.772,-60.211,-178.286,7.083,148.821
C06786=1152.445,179.523,-60.189,-178.288,7.082,148.822
C06787=1152.450,179.275,-60.166,-178.291,7.080,148.822
C06788=1152.455,179.026,-60.143,-178.294,7.077,148.822
C06789=1152.459,178.777,-60.120,-178.297,7.075,148.822
C06790=1152.464,178.527,-60.097,-178.299,7.072,148.823
C06791=1152.468,178.279,-60.075,-178.302,7.071,148.823
C06792=1152.473,178.030,-60.051,-178.305,7.069,148.823
C06793=1152.477,177.781,-60.029,-178.308,7.066,148.824
C06794=1152.482,177.532,-60.006,-178.310,7.064,148.824
C06795=1152.486,177.284,-59.984,-178.313,7.063,148.824
C06796=1152.491,177.034,-59.961,-178.316,7.060,148.825
C06797=1152.495,176.785,-59.938,-178.318,7.058,148.825
C06798=1152.500,176.536,-59.916,-178.321,7.056,148.825
C06799=1152.505,176.288,-59.893,-178.324,7.054,148.825
C06800=1152.510,176.039,-59.870,-178.327,7.052,148.826
C06801=1152.514,175.789,-59.848,-178.330,7.049,148.826
C06802=1152.519,175.541,-59.825,-178.333,7.047,148.826
C06803=1152.524,175.292,-59.803,-178.335,7.045,148.827
C06804=1152.528,175.043,-59.779,-178.338,7.043,148.827
C06805=1152.533,174.794,-59.758,-178.341,7.041,148.827
C06806=1152.538,174.545,-59.734,-178.344,7.039,148.827
C06807=1152.542,174.296,-59.712,-178.347,7.037,148.828
C06808=1152.547,174.047,-59.689,-178.349,7.034,148.828
C06809=1152.552,173.798,-59.667,-178.352,7.033,148.828
C06810=1152.556,173.549,-59.644,-178.355,7.030,148.829
C06811=1152.561,173.300,-59.622,-178.358,7.028,148.829
C06812=1152.565,173.051,-59.600,-178.360,7.026,148.829
C06813=1152.570,172.802,-59.577,-178.363,7.024,148.830
C06814=1152.575,172.553,-59.555,-178.366,7.022,148.830
C06815=1152.579,172.305,-59.532,-178.369,7.020,148.830
C06816=1152.585,172.056,-59.510,-178.371,7.017,148.830
C06817=1152.589,171.806,-59.488,-178.374,7.016,148.831
C06818=1152.593,171.558,-59.465,-178.377,7.014,148.831
C06819=1152.598,171.309,-59.443,-178.380,7.011,148.831
C06820=1152.603,171.059,-59.421,-178.382,7.009,148.832
C06821=1152.607,170.811,-59.398,-178.385,7.008,148.832
C06822=1152.612,170.562,-59.376,-178.388,7.006,148.832
C06823=1152.617,170.312,-59.354,-178.391,7.003,148.833
C06824=1152.621,170.064,-59.331,-178.393,7.001,148.833
C06825=1152.626,169.815,-59.309,-178.396,6.999,148.833
C06826=1152.631,169.566,-59.287,-178.399,6.997,148.834
C06827=1152.635,169.317,-59.265,-178.402,6.995,148.834
C06828=1152.640,169.069,-59.243,-178.404,6.993,148.834
C06829=1152.645,168.819,-59.220,-178.407,6.990,148.834
C06830=1152.649,168.570,-59.198,-178.410,6.989,148.835
C06831=1152.654,168.321,-59.176,-178.413,6.987,148.835
C06832=1152.658,168.072,-59.154,-178.415,6.985,148.836
C06833=1152.664,167.823,-59.131,-178.418,6.982,148.836
C06834=1152.668,167.574,-59.109,-178.421,6.981,148.836
C06835=1152.673,167.325,-59.087,-178.424,6.979,148.836
C06836=1152.677,167.076,-59.065,-178.427,6.976,148.837
C06837=1152.683,166.827,-59.043,-178.430,6.975,148.837
C06838=1152.687,166.578,-59.021,-178.432,6.973,148.837
C06839=1152.692,166.329,-58.999,-178.435,6.971,148.838
C06840=1152.696,166.080,-58.977,-178.438,6.968,148.838
C06841=1152.701,165.831,-58.956,-178.441,6.966,148.838
C06842=1152.705,165.582,-58.933,-178.443,6.965,148.839
C06843=1152.710,165.333,-58.911,-178.446,6.962,148.839
C06844=1152.715,165.084,-58.889,-178.449,6.960,148.839
C06845=1152.720,164.835,-58.867,-178.451,6.958,148.840
C06846=1152.724,164.586,-58.845,-178.454,6.957,148.840
C06847=1152.729,164.337,-58.823,-178.457,6.954,148.840
C06848=1152.733,164.088,-58.801,-178.460,6.952,148.841
C06849=1152.738,163.839,-58.779,-178.462,6.950,148.841
C06850=1152.743,163.591,-58.758,-178.465,6.949,148.841
C06851=1152.747,163.342,-58.736,-178.468,6.946,148.842
C06852=1152.752,163.093,-58.714,-178.471,6.944,148.842
C06853=1152.756,162.844,-58.692,-178.474,6.943,148.842
C06854=1152.762,162.594,-58.670,-178.476,6.940,148.843
C06855=1152.766,162.345,-58.648,-178.479,6.938,148.843
C06856=1152.771,162.096,-58.627,-178.482,6.936,148.843
C06857=1152.776,161.847,-58.605,-178.485,6.934,148.844
C06858=1152.780,161.598,-58.583,-178.487,6.933,148.844
C06859=1152.785,161.349,-58.561,-178.490,6.930,148.844
C06860=1152.789,161.100,-58.539,-178.493,6.928,148.845
C06861=1152.794,160.851,-58.518,-178.496,6.926,148.845
C06862=1152.799,160.602,-58.497,-178.498,6.925,148.845
C06863=1152.804,160.353,-58.475,-178.502,6.922,148.846
C06864=1152.809,160.104,-58.453,-178.504,6.920,148.846
C06865=1152.813,159.855,-58.431,-178.507,6.919,148.846
C06866=1152.818,159.606,-58.409,-178.509,6.917,148.847
C06867=1152.823,159.357,-58.388,-178.512,6.914,148.847
C06868=1152.827,159.108,-58.366,-178.515,6.912,148.847
C06869=1152.831,158.859,-58.345,-178.518,6.911,148.848
C06870=1152.836,158.611,-58.323,-178.521,6.909,148.848
C06871=1152.841,158.361,-58.302,-178.523,6.907,148.848
C06872=1152.846,158.092,-58.278,-178.527,6.905,148.849
C06873=1152.851,157.823,-58.255,-178.529,6.903,148.849
C06874=1152.857,157.554,-58.232,-178.533,6.900,148.850
C06875=1152.861,157.286,-58.209,-178.535,6.898,148.850
C06876=1152.866,157.036,-58.187,-178.538,6.897,148.850
C06877=1152.871,156.787,-58.166,-178.541,6.894,148.850
C06878=1152.876,156.539,-58.144,-178.543,6.892,148.851
C06879=1152.880,156.289,-58.123,-178.546,6.890,148.851
C06880=1152.885,156.040,-58.101,-178.549,6.889,148.852
C06881=1152.890,155.791,-58.080,-178.552,6.887,148.852
C06882=1152.894,155.542,-58.059,-178.555,6.884,148.852
C06883=1152.899,155.293,-58.037,-178.558,6.883,148.853
C06884=1152.904,155.044,-58.016,-178.560,6.881,148.853
C06885=1152.909,154.795,-57.994,-178.562,6.879,148.853
C06886=1152.913,154.545,-57.973,-178.565,6.877,148.854
C06887=1152.917,154.297,-57.952,-178.568,6.875,148.854
C06888=1152.922,154.048,-57.931,-178.571,6.873,148.854
C06889=1152.927,153.799,-57.909,-178.574,6.871,148.855
C06890=1152.932,153.549,-57.888,-178.577,6.869,148.855
C06891=1152.937,153.300,-57.866,-178.579,6.868,148.855
C06892=1152.941,153.051,-57.846,-178.583,6.865,148.856
C06893=1152.946,152.803,-57.824,-178.585,6.863,148.856
C06894=1152.951,152.553,-57.803,-178.588,6.862,148.857
C06895=1152.956,152.304,-57.781,-178.590,6.860,148.857
C06896=1152.960,152.055,-57.761,-178.593,6.858,148.857
C06897=1152.965,151.807,-57.739,-178.596,6.856,148.858
C06898=1152.970,151.557,-57.718,-178.599,6.854,148.858
C06899=1152.974,151.308,-57.698,-178.602,6.852,148.858
C06900=1152.979,151.059,-57.676,-178.604,6.850,148.859
C06901=1152.984,150.810,-57.655,-178.607,6.848,148.859
C06902=1152.989,150.561,-57.633,-178.610,6.847,148.859
C06903=1152.993,150.312,-57.613,-178.612,6.845,148.860
C06904=1152.998,150.063,-57.592,-178.616,6.842,148.860
C06905=1153.003,149.813,-57.570,-178.618,6.841,148.861
C06906=1153.007,149.565,-57.549,-178.621,6.839,148.861
C06907=1153.012,149.315,-57.528,-178.623,6.837,148.861
C06908=1153.017,149.067,-57.507,-178.626,6.835,148.861
C06909=1153.022,148.818,-57.486,-178.629,6.833,148.862
C06910=1153.027,148.568,-57.465,-178.631,6.832,148.862
C06911=1153.031,148.319,-57.445,-178.635,6.829,148.863
C06912=1153.035,148.070,-57.423,-178.637,6.827,148.863
C06913=1153.041,147.821,-57.402,-178.640,6.826,148.863
C06914=1153.045,147.572,-57.381,-178.643,6.824,148.864
C06915=1153.050,147.323,-57.361,-178.646,6.822,148.864
C06916=1153.055,147.074,-57.340,-178.648,6.821,148.865
C06917=1153.060,146.825,-57.318,-178.651,6.819,148.865
C06918=1153.064,146.576,-57.298,-178.654,6.816,148.865
C06919=1153.069,146.327,-57.277,-178.657,6.815,148.866
C06920=1153.074,146.078,-57.256,-178.660,6.813,148.866
C06921=1153.078,145.828,-57.235,-178.662,6.811,148.866
C06922=1153.083,145.579,-57.214,-178.665,6.809,148.867
C06923=1153.087,145.330,-57.193,-178.668,6.808,148.867
C06924=1153.093,145.081,-57.172,-178.670,6.806,148.867
C06925=1153.097,144.832,-57.152,-178.673,6.804,148.868
C06926=1153.102,144.583,-57.131,-178.675,6.802,148.868
C06927=1153.107,144.334,-57.111,-178.679,6.800,148.869
C06928=1153.112,144.085,-57.090,-178.681,6.798,148.869
C06929=1153.116,143.836,-57.069,-178.684,6.796,148.869
C06930=1153.121,143.587,-57.048,-178.687,6.794,148.870
C06931=1153.126,143.338,-57.028,-178.690,6.793,148.870
C06932=1153.130,143.089,-57.008,-178.692,6.791,148.870
C06933=1153.135,142.839,-56.987,-178.695,6.789,148.871
C06934=1153.140,142.590,-56.966,-178.698,6.788,148.871
C06935=1153.145,142.341,-56.945,-178.700,6.786,148.872
C06936=1153.150,142.092,-56.925,-178.704,6.783,148.872
C06937=1153.155,141.843,-56.904,-178.706,6.782,148.872
C06938=1153.159,141.594,-56.884,-178.709,6.780,148.873
C06939=1153.164,141.345,-56.863,-178.712,6.778,148.873
C06940=1153.169,141.096,-56.842,-178.715,6.776,148.874
C06941=1153.173,140.847,-56.822,-178.717,6.775,148.874
C06942=1153.178,140.598,-56.802,-178.720,6.773,148.874
C06943=1153.183,140.349,-56.781,-178.723,6.771,148.875
C06944=1153.187,140.100,-56.760,-178.725,6.770,148.875
C06945=1153.192,139.850,-56.739,-178.728,6.768,148.875
C06946=1153.197,139.601,-56.720,-178.731,6.766,148.876
C06947=1153.202,139.352,-56.699,-178.734,6.764,148.876
C06948=1153.207,139.103,-56.678,-178.736,6.763,148.877
C06949=1153.211,138.854,-56.658,-178.740,6.760,148.877
C06950=1153.216,138.605,-56.637,-178.742,6.758,148.877
C06951=1153.220,138.356,-56.617,-178.745,6.757,148.878
C06952=1153.226,138.106,-56.597,-178.748,6.755,148.878
C06953=1153.230,137.857,-56.576,-178.750,6.753,148.879
C06954=1153.234,137.608,-56.556,-178.753,6.752,148.879
C06955=1153.240,137.359,-56.535,-178.756,6.750,148.879
C06956=1153.244,137.109,-56.516,-178.759,6.748,148.880
C06957=1153.249,136.860,-56.495,-178.761,6.746,148.880
C06958=1153.253,136.611,-56.475,-178.764,6.745,148.881
C06959=1153.259,136.363,-56.454,-178.767,6.743,148.881
C06960=1153.264,136.113,-56.435,-178.769,6.741,148.881
C06961=1153.268,135.864,-56.414,-178.772,6.740,148.882
C06962=1153.273,135.615,-56.394,-178.775,6.738,148.882
C06963=1153.278,135.365,-56.374,-178.777,6.736,148.882
C06964=1153.283,135.116,-56.353,-178.780,6.734,148.883
C06965=1153.287,134.867,-56.333,-178.783,6.733,148.883
C06966=1153.292,134.618,-56.313,-178.786,6.731,148.884
C06967=1153.296,134.369,-56.293,-178.789,6.728,148.884
C06968=1153.302,134.120,-56.272,-178.792,6.727,148.884
C06969=1153.307,133.871,-56.252,-178.794,6.725,148.885
C06970=1153.311,133.622,-56.232,-178.797,6.723,148.885
C06971=1153.316,133.372,-56.212,-178.800,6.722,148.886
C06972=1153.320,133.123,-56.192,-178.802,6.720,148.886
C06973=1153.325,132.874,-56.172,-178.805,6.718,148.886
C06974=1153.330,132.626,-56.152,-178.808,6.717,148.887
C06975=1153.335,132.376,-56.131,-178.811,6.715,148.887
C06976=1153.340,132.108,-56.110,-178.814,6.713,148.888
C06977=1153.345,131.839,-56.089,-178.817,6.712,148.888
C06978=1153.350,131.571,-56.067,-178.820,6.709,148.889
C06979=1153.355,131.302,-56.046,-178.823,6.707,148.889
C06980=1153.360,131.052,-56.026,-178.825,6.706,148.889
C06981=1153.365,130.803,-56.006,-178.828,6.704,148.890
C06982=1153.370,130.554,-55.986,-178.831,6.703,148.890
C06983=1153.375,130.305,-55.966,-178.834,6.701,148.891
C06984=1153.380,130.056,-55.946,-178.837,6.699,148.891
C06985=1153.384,129.807,-55.925,-178.839,6.698,148.892
C06986=1153.389,129.557,-55.906,-178.842,6.696,148.892
C06987=1153.394,129.309,-55.886,-178.845,6.694,148.892
C06988=1153.399,129.059,-55.866,-178.847,6.692,148.893
C06989=1153.403,128.810,-55.847,-178.850,6.691,148.893
C06990=1153.408,128.561,-55.826,-178.853,6.689,148.894
C06991=1153.413,128.312,-55.807,-178.856,6.687,148.894
C06992=1153.418,128.063,-55.787,-178.858,6.686,148.894
C06993=1153.422,127.814,-55.767,-178.861,6.684,148.895
C06994=1153.427,127.564,-55.747,-178.864,6.682,148.895
C06995=1153.433,127.315,-55.728,-178.866,6.680,148.896
C06996=1153.437,127.066,-55.707,-178.869,6.679,148.896
C06997=1153.442,126.817,-55.688,-178.872,6.677,148.897
C06998=1153.446,126.567,-55.668,-178.875,6.676,148.897
C06999=1153.452,126.319,-55.648,-178.878,6.674,148.897
C07000=1153.456,126.070,-55.629,-178.881,6.672,148.898
C07001=1153.460,125.820,-55.609,-178.883,6.670,148.898
C07002=1153.466,125.571,-55.590,-178.886,6.669,148.899
C07003=1153.470,125.322,-55.570,-178.889,6.667,148.899
C07004=1153.475,125.073,-55.550,-178.891,6.665,148.899
C07005=1153.480,124.824,-55.531,-178.894,6.664,148.900
C07006=1153.485,124.574,-55.511,-178.896,6.663,148.900
C07007=1153.490,124.325,-55.492,-178.899,6.661,148.901
C07008=1153.495,124.076,-55.472,-178.902,6.660,148.901
C07009=1153.499,123.827,-55.452,-178.905,6.658,148.902
C07010=1153.503,123.577,-55.433,-178.908,6.656,148.902
C07011=1153.509,123.329,-55.414,-178.910,6.655,148.902
C07012=1153.513,123.079,-55.394,-178.913,6.653,148.903
C07013=1153.518,122.829,-55.374,-178.916,6.651,148.903
C07014=1153.524,122.581,-55.355,-178.918,6.649,148.904
C07015=1153.528,122.331,-55.335,-178.921,6.648,148.904
C07016=1153.532,122.082,-55.315,-178.924,6.646,148.904
C07017=1153.537,121.834,-55.296,-178.927,6.644,148.905
C07018=1153.542,121.584,-55.277,-178.930,6.643,148.905
C07019=1153.547,121.335,-55.257,-178.933,6.641,148.906
C07020=1153.551,121.086,-55.238,-178.935,6.640,148.906
C07021=1153.556,120.836,-55.219,-178.938,6.638,148.907
C07022=1153.562,120.587,-55.199,-178.941,6.636,148.907
C07023=1153.566,120.338,-55.180,-178.943,6.634,148.907
C07024=1153.572,120.089,-55.160,-178.946,6.634,148.908
C07025=1153.576,119.840,-55.141,-178.948,6.632,148.908
C07026=1153.580,119.590,-55.122,-178.951,6.630,148.909
C07027=1153.586,119.341,-55.102,-178.954,6.629,148.909
C07028=1153.590,119.092,-55.083,-178.957,6.627,148.910
C07029=1153.595,118.843,-55.064,-178.960,6.625,148.910
C07030=1153.600,118.594,-55.044,-178.962,6.624,148.910
C07031=1153.605,118.345,-55.025,-178.965,6.622,148.911
C07032=1153.609,118.095,-55.007,-178.968,6.620,148.911
C07033=1153.614,117.845,-54.987,-178.970,6.619,148.912
C07034=1153.620,117.596,-54.968,-178.974,6.617,148.912
C07035=1153.624,117.347,-54.949,-178.976,6.616,148.913
C07036=1153.629,117.098,-54.929,-178.979,6.614,148.913
C07037=1153.634,116.849,-54.910,-178.981,6.613,148.913
C07038=1153.638,116.600,-54.891,-178.984,6.611,148.914
C07039=1153.643,116.351,-54.871,-178.987,6.610,148.914
C07040=1153.649,116.101,-54.853,-178.989,6.608,148.915
C07041=1153.653,115.852,-54.834,-178.993,6.606,148.915
C07042=1153.658,115.603,-54.814,-178.995,6.605,148.916
C07043=1153.663,115.353,-54.795,-178.998,6.603,148.916
C07044=1153.667,115.105,-54.776,-179.001,6.601,148.917
C07045=1153.672,114.855,-54.757,-179.003,6.600,148.917
C07046=1153.677,114.606,-54.738,-179.006,6.599,148.917
C07047=1153.682,114.357,-54.719,-179.008,6.597,148.918
C07048=1153.686,114.108,-54.700,-179.012,6.596,148.918
C07049=1153.691,113.858,-54.681,-179.014,6.594,148.919
C07050=1153.697,113.609,-54.662,-179.017,6.592,148.919
C07051=1153.701,113.360,-54.643,-179.020,6.591,148.920
C07052=1153.706,113.110,-54.624,-179.022,6.589,148.920
C07053=1153.711,112.862,-54.606,-179.025,6.587,148.920
C07054=1153.716,112.612,-54.586,-179.028,6.586,148.921
C07055=1153.721,112.363,-54.568,-179.030,6.585,148.921
C07056=1153.725,112.113,-54.548,-179.033,6.583,148.922
C07057=1153.730,111.865,-54.530,-179.036,6.582,148.922
C07058=1153.735,111.615,-54.511,-179.039,6.580,148.923
C07059=1153.740,111.366,-54.492,-179.041,6.578,148.923
C07060=1153.745,111.117,-54.473,-179.045,6.577,148.924
C07061=1153.749,110.867,-54.454,-179.047,6.575,148.924
C07062=1153.755,110.618,-54.435,-179.049,6.574,148.925
C07063=1153.759,110.369,-54.417,-179.052,6.573,148.925
C07064=1153.764,110.120,-54.397,-179.055,6.571,148.925
C07065=1153.769,109.871,-54.379,-179.058,6.569,148.926
C07066=1153.774,109.621,-54.360,-179.061,6.568,148.926
C07067=1153.779,109.372,-54.341,-179.064,6.566,148.927
C07068=1153.784,109.122,-54.322,-179.066,6.564,148.927
C07069=1153.788,108.874,-54.303,-179.068,6.564,148.928
C07070=1153.793,108.624,-54.285,-179.071,6.562,148.928
C07071=1153.798,108.375,-54.266,-179.074,6.560,148.929
C07072=1153.803,108.126,-54.248,-179.077,6.559,148.929
C07073=1153.808,107.877,-54.228,-179.080,6.557,148.929
C07074=1153.812,107.627,-54.210,-179.082,6.555,148.930
C07075=1153.817,107.378,-54.192,-179.085,6.554,148.930
C07076=1153.823,107.129,-54.173,-179.088,6.553,148.931
C07077=1153.827,106.879,-54.154,-179.091,6.551,148.931
C07078=1153.832,106.631,-54.136,-179.093,6.550,148.932
C07079=1153.837,106.381,-54.117,-179.096,6.548,148.932
C07080=1153.842,106.112,-54.097,-179.099,6.546,148.933
C07081=1153.847,105.844,-54.077,-179.102,6.545,148.933
C07082=1153.852,105.576,-54.057,-179.105,6.543,148.934
C07083=1153.858,105.307,-54.037,-179.108,6.542,148.934
C07084=1153.862,105.058,-54.018,-179.111,6.540,148.935
C07085=1153.867,104.809,-54.000,-179.113,6.539,148.935
C07086=1153.873,104.559,-53.982,-179.115,6.538,148.935
C07087=1153.877,104.311,-53.963,-179.118,6.536,148.936
C07088=1153.882,104.061,-53.945,-179.121,6.535,148.937
C07089=1153.887,103.811,-53.926,-179.124,6.533,148.937
C07090=1153.892,103.563,-53.907,-179.127,6.531,148.937
C07091=1153.896,103.313,-53.889,-179.130,6.530,148.938
C07092=1153.901,103.064,-53.871,-179.132,6.529,148.938
C07093=1153.907,102.814,-53.852,-179.135,6.527,148.939
C07094=1153.911,102.566,-53.834,-179.138,6.526,148.939
C07095=1153.916,102.316,-53.815,-179.140,6.524,148.940
C07096=1153.921,102.067,-53.797,-179.143,6.522,148.940
C07097=1153.926,101.818,-53.779,-179.146,6.522,148.941
C07098=1153.931,101.568,-53.761,-179.148,6.520,148.941
C07099=1153.935,101.319,-53.742,-179.151,6.518,148.942
C07100=1153.940,101.070,-53.724,-179.154,6.517,148.942
C07101=1153.945,100.820,-53.706,-179.157,6.515,148.943
C07102=1153.950,100.571,-53.688,-179.159,6.514,148.943
C07103=1153.956,100.322,-53.669,-179.162,6.513,148.943
C07104=1153.960,100.072,-53.651,-179.165,6.511,148.944
C07105=1153.964,99.823,-53.632,-179.167,6.509,148.944
C07106=1153.969,99.574,-53.614,-179.170,6.509,148.945
C07107=1153.974,99.325,-53.596,-179.173,6.507,148.945
C07108=1153.979,99.076,-53.578,-179.175,6.506,148.946
C07109=1153.984,98.826,-53.559,-179.178,6.504,148.946
C07110=1153.989,98.576,-53.541,-179.181,6.502,148.947
C07111=1153.994,98.327,-53.523,-179.184,6.502,148.947
C07112=1153.999,98.078,-53.505,-179.186,6.500,148.948
C07113=1154.004,97.829,-53.487,-179.189,6.498,148.948
C07114=1154.009,97.580,-53.470,-179.192,6.497,148.949
C07115=1154.013,97.330,-53.451,-179.194,6.496,148.949
C07116=1154.018,97.081,-53.433,-179.197,6.494,148.949
C07117=1154.023,96.832,-53.415,-179.200,6.493,148.950
C07118=1154.028,96.582,-53.397,-179.203,6.491,148.951
C07119=1154.033,96.333,-53.379,-179.205,6.490,148.951
C07120=1154.038,96.084,-53.361,-179.208,6.489,148.951
C07121=1154.043,95.835,-53.343,-179.211,6.487,148.952
C07122=1154.048,95.585,-53.324,-179.214,6.486,148.952
C07123=1154.053,95.335,-53.306,-179.216,6.485,148.953
C07124=1154.057,95.086,-53.288,-179.219,6.483,148.953
C07125=1154.062,94.837,-53.270,-179.221,6.481,148.954
C07126=1154.067,94.588,-53.252,-179.225,6.480,148.954
C07127=1154.072,94.339,-53.234,-179.227,6.479,148.955
C07128=1154.077,94.090,-53.216,-179.230,6.478,148.955
C07129=1154.082,93.840,-53.198,-179.232,6.476,148.956
C07130=1154.087,93.591,-53.181,-179.235,6.475,148.956
C07131=1154.092,93.341,-53.163,-179.238,6.474,148.957
C07132=1154.096,93.092,-53.145,-179.240,6.472,148.957
C07133=1154.101,92.842,-53.127,-179.243,6.470,148.957
C07134=1154.106,92.593,-53.109,-179.246,6.469,148.958
C07135=1154.110,92.344,-53.092,-179.248,6.468,148.959
C07136=1154.115,92.095,-53.074,-179.251,6.466,148.959
C07137=1154.121,91.845,-53.056,-179.254,6.465,148.960
C07138=1154.126,91.596,-53.038,-179.256,6.464,148.960
C07139=1154.130,91.347,-53.020,-179.259,6.463,148.960
C07140=1154.135,91.098,-53.002,-179.262,6.461,148.961
C07141=1154.141,90.848,-52.985,-179.265,6.460,148.962
C07142=1154.145,90.599,-52.967,-179.267,6.459,148.962
C07143=1154.150,90.350,-52.949,-179.270,6.457,148.962
C07144=1154.155,90.101,-52.931,-179.273,6.455,148.963
C07145=1154.160,89.851,-52.914,-179.276,6.454,148.963
C07146=1154.165,89.602,-52.897,-179.278,6.453,148.964
C07147=1154.170,89.353,-52.879,-179.281,6.451,148.964
C07148=1154.175,89.103,-52.861,-179.284,6.450,148.965
C07149=1154.180,88.854,-52.843,-179.286,6.449,148.965
C07150=1154.185,88.605,-52.825,-179.289,6.447,148.966
C07151=1154.190,88.355,-52.808,-179.292,6.446,148.966
C07152=1154.194,88.106,-52.791,-179.294,6.445,148.967
C07153=1154.199,87.857,-52.773,-179.297,6.444,148.967
C07154=1154.204,87.607,-52.755,-179.300,6.442,148.968
C07155=1154.209,87.358,-52.737,-179.303,6.441,148.968
C07156=1154.214,87.109,-52.719,-179.305,6.440,148.969
C07157=1154.218,86.859,-52.703,-179.308,6.438,148.969
C07158=1154.223,86.610,-52.685,-179.311,6.437,148.970
C07159=1154.229,86.360,-52.668,-179.313,6.436,148.970
C07160=1154.234,86.111,-52.650,-179.316,6.434,148.971
C07161=1154.239,85.861,-52.632,-179.319,6.432,148.971
C07162=1154.243,85.612,-52.615,-179.321,6.432,148.972
C07163=1154.248,85.363,-52.597,-179.324,6.430,148.972
C07164=1154.253,85.113,-52.580,-179.327,6.429,148.973
C07165=1154.258,84.864,-52.562,-179.329,6.428,148.973
C07166=1154.263,84.615,-52.545,-179.332,6.426,148.974
C07167=1154.268,84.366,-52.527,-179.335,6.425,148.974
C07168=1154.273,84.116,-52.510,-179.338,6.424,148.975
C07169=1154.277,83.868,-52.493,-179.340,6.423,148.975
C07170=1154.283,83.618,-52.475,-179.343,6.421,148.976
C07171=1154.288,83.368,-52.458,-179.345,6.420,148.976
C07172=1154.292,83.119,-52.441,-179.348,6.419,148.977
C07173=1154.297,82.869,-52.424,-179.351,6.417,148.977
C07174=1154.302,82.620,-52.406,-179.353,6.416,148.978
C07175=1154.307,82.371,-52.389,-179.356,6.415,148.978
C07176=1154.312,82.122,-52.371,-179.359,6.413,148.979
C07177=1154.317,81.872,-52.354,-179.361,6.412,148.979
C07178=1154.322,81.623,-52.337,-179.365,6.411,148.980
C07179=1154.327,81.374,-52.319,-179.367,6.409,148.980
C07180=1154.332,81.124,-52.302,-179.369,6.408,148.981
C07181=1154.336,80.874,-52.285,-179.373,6.407,148.981
C07182=1154.341,80.625,-52.267,-179.375,6.405,148.982
C07183=1154.347,80.376,-52.251,-179.378,6.405,148.982
C07184=1154.352,80.108,-52.232,-179.381,6.403,148.983
C07185=1154.357,79.839,-52.214,-179.383,6.402,148.983
C07186=1154.363,79.571,-52.195,-179.387,6.400,148.984
C07187=1154.367,79.303,-52.177,-179.389,6.399,148.984
C07188=1154.373,79.053,-52.159,-179.392,6.398,148.985
C07189=1154.377,78.803,-52.143,-179.395,6.396,148.985
C07190=1154.383,78.555,-52.125,-179.397,6.395,148.986
C07191=1154.387,78.305,-52.108,-179.400,6.394,148.986
C07192=1154.392,78.056,-52.091,-179.403,6.393,148.987
C07193=1154.398,77.806,-52.074,-179.405,6.392,148.987
C07194=1154.402,77.557,-52.057,-179.408,6.390,148.988
C07195=1154.408,77.308,-52.040,-179.411,6.389,148.988
C07196=1154.412,77.058,-52.023,-179.413,6.388,148.989
C07197=1154.417,76.809,-52.006,-179.416,6.386,148.989
C07198=1154.422,76.559,-51.989,-179.419,6.386,148.990
C07199=1154.428,76.310,-51.972,-179.421,6.384,148.990
C07200=1154.432,76.061,-51.955,-179.424,6.383,148.991
C07201=1154.437,75.811,-51.937,-179.427,6.382,148.991
C07202=1154.441,75.562,-51.921,-179.429,6.380,148.992
C07203=1154.447,75.312,-51.904,-179.433,6.379,148.992
C07204=1154.452,75.063,-51.887,-179.435,6.378,148.993
C07205=1154.456,74.814,-51.871,-179.437,6.376,148.993
C07206=1154.461,74.564,-51.853,-179.440,6.376,148.994
C07207=1154.467,74.315,-51.837,-179.443,6.374,148.994
C07208=1154.471,74.066,-51.819,-179.446,6.372,148.995
C07209=1154.476,73.817,-51.802,-179.448,6.372,148.995
C07210=1154.481,73.567,-51.785,-179.451,6.370,148.996
C07211=1154.486,73.318,-51.769,-179.453,6.369,148.996
C07212=1154.491,73.068,-51.752,-179.456,6.368,148.997
C07213=1154.496,72.819,-51.735,-179.459,6.366,148.997
C07214=1154.501,72.570,-51.719,-179.462,6.366,148.998
C07215=1154.506,72.320,-51.701,-179.464,6.364,148.998
C07216=1154.511,72.071,-51.685,-179.467,6.363,148.999
C07217=1154.515,71.821,-51.668,-179.470,6.362,149.000
C07218=1154.521,71.572,-51.651,-179.472,6.361,149.000
C07219=1154.525,71.323,-51.634,-179.475,6.359,149.000
C07220=1154.530,71.073,-51.618,-179.478,6.358,149.001
C07221=1154.536,70.824,-51.601,-179.480,6.357,149.001
C07222=1154.540,70.574,-51.584,-179.483,6.356,149.002
C07223=1154.545,70.325,-51.567,-179.485,6.355,149.003
C07224=1154.551,70.075,-51.551,-179.488,6.353,149.003
C07225=1154.555,69.826,-51.535,-179.491,6.353,149.004
C07226=1154.560,69.576,-51.518,-179.494,6.351,149.004
C07227=1154.566,69.327,-51.501,-179.496,6.350,149.005
C07228=1154.570,69.078,-51.484,-179.499,6.349,149.005
C07229=1154.575,68.829,-51.468,-179.502,6.347,149.006
C07230=1154.580,68.579,-51.451,-179.504,6.347,149.006
C07231=1154.585,68.330,-51.434,-179.507,6.345,149.007
C07232=1154.590,68.080,-51.419,-179.509,6.344,149.007
C07233=1154.595,67.831,-51.402,-179.512,6.343,149.008
C07234=1154.600,67.581,-51.385,-179.515,6.341,149.008
C07235=1154.605,67.332,-51.368,-179.517,6.341,149.009
C07236=1154.610,67.083,-51.352,-179.521,6.339,149.009
C07237=1154.615,66.834,-51.335,-179.523,6.338,149.010
C07238=1154.620,66.584,-51.319,-179.525,6.337,149.010
C07239=1154.625,66.334,-51.302,-179.528,6.336,149.011
C07240=1154.630,66.085,-51.286,-179.531,6.335,149.011
C07241=1154.634,65.836,-51.269,-179.533,6.334,149.012
C07242=1154.640,65.586,-51.254,-179.536,6.332,149.012
C07243=1154.645,65.337,-51.236,-179.538,6.332,149.013
C07244=1154.649,65.087,-51.220,-179.542,6.330,149.013
C07245=1154.654,64.838,-51.203,-179.544,6.329,149.014
C07246=1154.659,64.588,-51.187,-179.546,6.328,149.014
C07247=1154.664,64.339,-51.171,-179.550,6.326,149.015
C07248=1154.669,64.090,-51.154,-179.552,6.326,149.015
C07249=1154.675,63.840,-51.138,-179.555,6.324,149.016
C07250=1154.679,63.591,-51.122,-179.557,6.323,149.017
C07251=1154.684,63.342,-51.105,-179.560,6.322,149.017
C07252=1154.689,63.092,-51.089,-179.563,6.321,149.018
C07253=1154.694,62.843,-51.073,-179.565,6.320,149.018
C07254=1154.699,62.593,-51.057,-179.567,6.319,149.019
C07255=1154.704,62.344,-51.041,-179.571,6.317,149.019
C07256=1154.709,62.095,-51.024,-179.573,6.317,149.020
C07257=1154.713,61.845,-51.008,-179.576,6.315,149.020
C07258=1154.719,61.595,-50.991,-179.578,6.314,149.021
C07259=1154.724,61.345,-50.975,-179.581,6.313,149.021
C07260=1154.729,61.097,-50.959,-179.584,6.312,149.022
C07261=1154.734,60.847,-50.942,-179.586,6.311,149.022
C07262=1154.739,60.598,-50.927,-179.589,6.310,149.023
C07263=1154.744,60.349,-50.910,-179.592,6.308,149.023
C07264=1154.749,60.099,-50.894,-179.594,6.308,149.024
C07265=1154.754,59.850,-50.878,-179.597,6.306,149.024
C07266=1154.759,59.600,-50.862,-179.599,6.305,149.025
C07267=1154.764,59.351,-50.846,-179.602,6.304,149.026
C07268=1154.769,59.101,-50.830,-179.605,6.303,149.026
C07269=1154.774,58.852,-50.814,-179.607,6.302,149.026
C07270=1154.778,58.602,-50.798,-179.610,6.301,149.027
C07271=1154.784,58.353,-50.781,-179.613,6.299,149.028
C07272=1154.788,58.103,-50.765,-179.615,6.299,149.028
C07273=1154.793,57.855,-50.749,-179.618,6.297,149.029
C07274=1154.799,57.605,-50.734,-179.620,6.296,149.029
C07275=1154.804,57.355,-50.718,-179.624,6.295,149.030
C07276=1154.809,57.106,-50.701,-179.626,6.294,149.030
C07277=1154.813,56.856,-50.685,-179.629,6.293,149.031
C07278=1154.818,56.607,-50.669,-179.631,6.292,149.031
C07279=1154.823,56.357,-50.653,-179.634,6.291,149.032
C07280=1154.829,56.108,-50.637,-179.636,6.290,149.032
C07281=1154.834,55.859,-50.621,-179.639,6.288,149.033
C07282=1154.839,55.609,-50.605,-179.642,6.288,149.033
C07283=1154.844,55.360,-50.590,-179.645,6.286,149.034
C07284=1154.848,55.110,-50.573,-179.647,6.286,149.035
C07285=1154.854,54.861,-50.557,-179.650,6.284,149.035
C07286=1154.859,54.611,-50.542,-179.652,6.283,149.035
C07287=1154.863,54.362,-50.526,-179.655,6.283,149.036
C07288=1154.868,54.094,-50.509,-179.658,6.281,149.037
C07289=1154.874,53.825,-50.492,-179.661,6.280,149.037
C07290=1154.880,53.557,-50.475,-179.663,6.279,149.038
C07291=1154.885,53.287,-50.457,-179.666,6.278,149.038
C07292=1154.890,53.038,-50.442,-179.669,6.276,149.039
C07293=1154.895,52.789,-50.426,-179.672,6.275,149.039
C07294=1154.900,52.539,-50.409,-179.674,6.275,149.040
C07295=1154.905,52.290,-50.394,-179.677,6.273,149.041
C07296=1154.910,52.041,-50.379,-179.679,6.272,149.041
C07297=1154.915,51.791,-50.363,-179.682,6.271,149.042
C07298=1154.920,51.541,-50.347,-179.684,6.270,149.042
C07299=1154.925,51.292,-50.331,-179.688,6.269,149.043
C07300=1154.930,51.042,-50.315,-179.690,6.268,149.043
C07301=1154.935,50.793,-50.299,-179.693,6.267,149.044
C07302=1154.940,50.544,-50.284,-179.695,6.266,149.044
C07303=1154.945,50.294,-50.269,-179.697,6.265,149.045
